KUKA KRL program: MyProgram_226().src

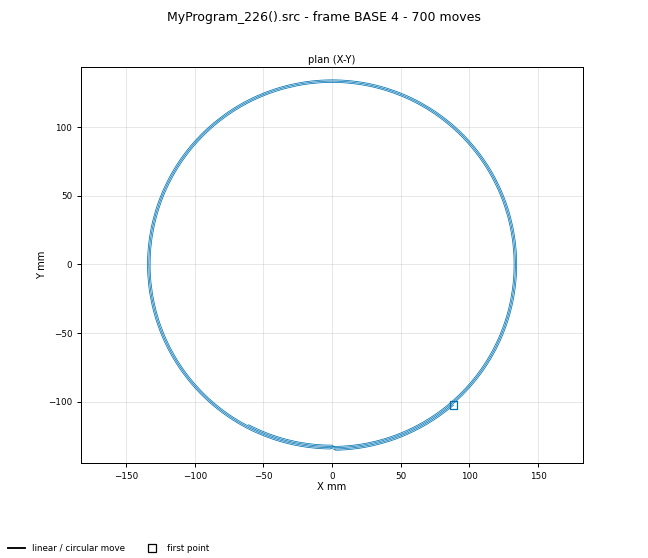
[picture p0: tool path of MyProgram_226().src in frame BASE 4, 700 of 700 moves have a stored position in this frame; points joined in program order, loops and branches not executed]
&ACCESS RVP
&REL 1
&PARAM TEMPLATE = C:\KRC\Roboter\Template\vorgabe
&PARAM EDITMASK = *
DEF MyProgram_226()
; ---- Setting reference (Base) ----
$BASE = BASE_DATA[4]

; --------------------------
; ---- Setting tool (TCP) ----
$TOOL = TOOL_DATA[3]
; --------------------------

$VEL.CP = VEL_APROX_PRINT
Startdeposition()
$VEL.CP = VEL_PRINT
LIN {X 88.4105,Y -102.4837,Z 156,A -52.8123,B 24.9683,C -1.3001,E1 25.1035,E2 499.4547} C_DIS
LIN {X 85.5901,Y -104.8506,Z 156,A -54.3172,B 24.9683,C -1.2995,E1 25.1003,E2 500.9552} C_DIS
LIN {X 81.9541,Y -107.7171,Z 156,A -56.2769,B 24.9686,C -1.2951,E1 25.096,E2 502.918} C_DIS
LIN {X 78.4285,Y -110.3106,Z 156,A -58.1174,B 24.9687,C -1.2919,E1 25.0918,E2 504.7597} C_DIS
LIN {X 75.1109,Y -112.5952,Z 156,A -59.7943,B 24.9688,C -1.2899,E1 25.0879,E2 506.4355} C_DIS
LIN {X 71.3717,Y -115.0019,Z 156,A -61.6528,B 24.969,C -1.2876,E1 25.0835,E2 508.2937} C_DIS
LIN {X 67.9053,Y -117.0821,Z 156,A -63.3421,B 24.969,C -1.2855,E1 25.0795,E2 509.9826} C_DIS
LIN {X 64.3345,Y -119.0819,Z 156,A -65.1517,B 24.9694,C -1.2782,E1 25.075,E2 511.8043} C_DIS
LIN {X 59.8875,Y -121.3766,Z 156,A -67.0719,B 24.9691,C -1.2855,E1 25.0703,E2 513.702} C_DIS
LIN {X 57.2409,Y -122.6479,Z 156,A -68.3239,B 24.9691,C -1.2829,E1 25.0671,E2 514.9567} C_DIS
LIN {X 53.5301,Y -124.3116,Z 156,A -70.0894,B 24.9694,C -1.2779,E1 25.0626,E2 516.7299} C_DIS
LIN {X 50.109,Y -125.7306,Z 156,A -71.756,B 24.9698,C -1.2701,E1 25.0582,E2 518.4109} C_DIS
LIN {X 45.2698,Y -127.5536,Z 156,A -73.8005,B 24.9696,C -1.275,E1 25.0529,E2 520.4396} C_DIS
LIN {X 42.4798,Y -128.5083,Z 156,A -75.0813,B 24.9697,C -1.2717,E1 25.0495,E2 521.7258} C_DIS
LIN {X 38.7522,Y -129.683,Z 156,A -76.6927,B 24.9697,C -1.272,E1 25.0452,E2 523.3335} C_DIS
LIN {X 33.3545,Y -131.173,Z 156,A -79.0675,B 24.9698,C -1.2692,E1 25.0388,E2 525.7112} C_DIS
LIN {X 30.1099,Y -131.9555,Z 156,A -80.5038,B 24.97,C -1.2665,E1 25.0349,E2 527.1518} C_DIS
LIN {X 26.6432,Y -132.6994,Z 156,A -82.044,B 24.9701,C -1.2631,E1 25.0307,E2 528.6983} C_DIS
LIN {X 22.4298,Y -133.4759,Z 156,A -83.877,B 24.9702,C -1.2605,E1 25.0256,E2 530.5353} C_DIS
LIN {X 18.3422,Y -134.1009,Z 156,A -85.6848,B 24.9704,C -1.2562,E1 25.0206,E2 532.3517} C_DIS
LIN {X 14.4718,Y -134.5715,Z 156,A -87.2354,B 24.9702,C -1.2606,E1 25.0163,E2 533.8908} C_DIS
LIN {X 10.295,Y -134.9561,Z 156,A -89.0367,B 24.9703,C -1.2583,E1 25.0113,E2 535.6965} C_DIS
LIN {X 6.6876,Y -135.1822,Z 156,A -90.5035,B 24.9703,C -1.261,E1 25.0072,E2 537.1563} C_DIS
LIN {X 2.7111,Y -135.3212,Z 156,A -92.2608,B 24.9704,C -1.2566,E1 25.0023,E2 538.9238} C_DIS
LIN {X 2.7111,Y -135.3212,Z 156,A -92.2608,B 24.9704,C -1.2566,E1 25.0023,E2 538.9238} C_DIS
Enddeposition()
LIN {X 0.9355,Y -134.409,Z 156,A -91.9033,B 23.562,C -1.0427,E1 23.5861,E2 538.9103} C_DIS
Startdeposition()
$VEL.CP = VEL_PRINT
LIN {X 4.9293,Y -134.3237,Z 156,A -90.1147,B 23.5618,C -1.0476,E1 23.5911,E2 537.11} C_DIS
LIN {X 8.6316,Y -134.1368,Z 156,A -88.4447,B 23.5616,C -1.0528,E1 23.5958,E2 535.4278} C_DIS
LIN {X 12.8622,Y -133.7968,Z 156,A -86.7417,B 23.5618,C -1.0483,E1 23.6005,E2 533.7369} C_DIS
LIN {X 17.0675,Y -133.3262,Z 156,A -84.913,B 23.5617,C -1.0507,E1 23.6056,E2 531.9039} C_DIS
LIN {X 20.2692,Y -132.8768,Z 156,A -83.6497,B 23.5619,C -1.0458,E1 23.609,E2 530.654} C_DIS
LIN {X 23.6425,Y -132.3179,Z 156,A -82.0981,B 23.5616,C -1.0517,E1 23.6133,E2 529.0893} C_DIS
LIN {X 27.7995,Y -131.5086,Z 156,A -80.2512,B 23.5615,C -1.0554,E1 23.6184,E2 527.2357} C_DIS
LIN {X 31.3885,Y -130.6971,Z 156,A -78.7676,B 23.5616,C -1.0525,E1 23.6224,E2 525.7614} C_DIS
LIN {X 37.2329,Y -129.1549,Z 156,A -76.2005,B 23.5616,C -1.0548,E1 23.6294,E2 523.193} C_DIS
LIN {X 41.5122,Y -127.844,Z 156,A -74.1617,B 23.5611,C -1.0638,E1 23.6348,E2 521.1358} C_DIS
LIN {X 45.1666,Y -126.5982,Z 156,A -72.4547,B 23.5609,C -1.0691,E1 23.6394,E2 519.4191} C_DIS
LIN {X 49.906,Y -124.8057,Z 156,A -70.4656,B 23.5612,C -1.0632,E1 23.6445,E2 517.4494} C_DIS
LIN {X 53.121,Y -123.4712,Z 156,A -69.0171,B 23.5612,C -1.0636,E1 23.6482,E2 516.0036} C_DIS
LIN {X 56.8828,Y -121.7847,Z 156,A -67.2053,B 23.5609,C -1.0692,E1 23.6528,E2 514.1828} C_DIS
LIN {X 60.3051,Y -120.1281,Z 156,A -65.5272,B 23.5607,C -1.0748,E1 23.657,E2 512.4955} C_DIS
LIN {X 63.8728,Y -118.27,Z 156,A -63.8371,B 23.5606,C -1.0765,E1 23.6612,E2 510.8063} C_DIS
LIN {X 67.8011,Y -116.0627,Z 156,A -61.9275,B 23.5605,C -1.0794,E1 23.6658,E2 508.8956} C_DIS
LIN {X 70.6321,Y -114.3619,Z 156,A -60.5125,B 23.5603,C -1.0824,E1 23.6692,E2 507.4778} C_DIS
LIN {X 74.425,Y -111.9304,Z 156,A -58.6117,B 23.5603,C -1.0852,E1 23.6737,E2 505.5767} C_DIS
LIN {X 78.0467,Y -109.4357,Z 156,A -56.7416,B 23.5601,C -1.0888,E1 23.6779,E2 503.7045} C_DIS
LIN {X 81.7345,Y -106.7094,Z 156,A -54.8243,B 23.56,C -1.091,E1 23.6822,E2 501.7892} C_DIS
LIN {X 85.2048,Y -103.9597,Z 156,A -53.1718,B 23.5603,C -1.0828,E1 23.6858,E2 500.1636} C_DIS
LIN {X 88.1779,Y -101.4502,Z 156,A -51.272,B 23.5596,C -1.0993,E1 23.6899,E2 498.2307} C_DIS
LIN {X 91.4896,Y -98.4739,Z 156,A -49.3955,B 23.5594,C -1.1027,E1 23.6937,E2 496.3539} C_DIS
LIN {X 94.6611,Y -95.4291,Z 156,A -47.7139,B 23.5597,C -1.0971,E1 23.697,E2 494.6937} C_DIS
LIN {X 97.4339,Y -92.597,Z 156,A -45.834,B 23.5591,C -1.1114,E1 23.7007,E2 492.7869} C_DIS
LIN {X 100.4874,Y -89.2739,Z 156,A -43.8982,B 23.5588,C -1.117,E1 23.7044,E2 490.8464} C_DIS
LIN {X 103.3752,Y -85.9131,Z 156,A -42.0362,B 23.5587,C -1.1205,E1 23.7077,E2 488.9846} C_DIS
LIN {X 105.5443,Y -83.234,Z 156,A -40.6446,B 23.5587,C -1.1203,E1 23.7101,E2 487.6004} C_DIS
LIN {X 108.2335,Y -79.7055,Z 156,A -38.3873,B 23.5575,C -1.1451,E1 23.714,E2 485.293} C_DIS
LIN {X 110.5538,Y -76.4555,Z 156,A -37.0233,B 23.5581,C -1.1318,E1 23.7161,E2 483.9693} C_DIS
LIN {X 112.6587,Y -73.3176,Z 156,A -35.4269,B 23.558,C -1.1356,E1 23.7185,E2 482.3719} C_DIS
LIN {X 115.0279,Y -69.5415,Z 156,A -33.5351,B 23.5577,C -1.1407,E1 23.7213,E2 480.4778} C_DIS
LIN {X 117.3269,Y -65.5891,Z 156,A -31.5842,B 23.5575,C -1.1465,E1 23.724,E2 478.5232} C_DIS
LIN {X 119.5762,Y -61.3894,Z 156,A -29.6624,B 23.5575,C -1.1468,E1 23.7265,E2 476.6115} C_DIS
LIN {X 121.1879,Y -58.1416,Z 156,A -28.1905,B 23.5575,C -1.1475,E1 23.7283,E2 475.1462} C_DIS
LIN {X 122.593,Y -55.1176,Z 156,A -26.9535,B 23.5577,C -1.142,E1 23.7297,E2 473.93} C_DIS
LIN {X 124.1713,Y -51.4639,Z 156,A -25.0102,B 23.5568,C -1.1604,E1 23.7319,E2 471.9523} C_DIS
LIN {X 125.5328,Y -48.0514,Z 156,A -23.4937,B 23.5568,C -1.1626,E1 23.7334,E2 470.4393} C_DIS
LIN {X 126.9947,Y -44.0372,Z 156,A -21.7357,B 23.5566,C -1.165,E1 23.7351,E2 468.6858} C_DIS
LIN {X 128.2984,Y -40.0882,Z 156,A -19.7977,B 23.5559,C -1.1795,E1 23.7367,E2 466.7237} C_DIS
LIN {X 129.3686,Y -36.4803,Z 156,A -18.3244,B 23.556,C -1.1776,E1 23.7379,E2 465.264} C_DIS
LIN {X 130.2418,Y -33.2273,Z 156,A -16.9031,B 23.5558,C -1.1815,E1 23.7389,E2 463.8419} C_DIS
LIN {X 131.0539,Y -29.8641,Z 156,A -15.439,B 23.5556,C -1.1856,E1 23.7398,E2 462.3765} C_DIS
LIN {X 131.8298,Y -26.2341,Z 156,A -13.7478,B 23.5551,C -1.1966,E1 23.7408,E2 460.6685} C_DIS
LIN {X 132.5689,Y -22.1919,Z 156,A -12.1079,B 23.5551,C -1.1963,E1 23.7416,E2 459.0396} C_DIS
LIN {X 133.1787,Y -18.1926,Z 156,A -10.3049,B 23.5547,C -1.2061,E1 23.7423,E2 457.2235} C_DIS
LIN {X 133.636,Y -14.4372,Z 156,A -8.8205,B 23.5547,C -1.2046,E1 23.7427,E2 455.7524} C_DIS
LIN {X 133.9718,Y -10.8981,Z 156,A -7.1925,B 23.5542,C -1.2155,E1 23.7431,E2 454.1074} C_DIS
LIN {X 134.2369,Y -6.8942,Z 156,A -5.5996,B 23.5542,C -1.2148,E1 23.7434,E2 452.5263} C_DIS
LIN {X 134.3785,Y -3.1364,Z 156,A -3.9402,B 23.5538,C -1.2231,E1 23.7435,E2 450.8569} C_DIS
LIN {X 134.4111,Y 0.902,Z 156,A -2.2554,B 23.5537,C -1.2268,E1 23.7435,E2 449.1737} C_DIS
LIN {X 134.3168,Y 5.1048,Z 156,A -0.5175,B 23.5535,C -1.2297,E1 23.7434,E2 447.4395} C_DIS
LIN {X 134.1212,Y 8.8838,Z 156,A 1.1946,B 23.553,C -1.2402,E1 23.7431,E2 445.7121} C_DIS
LIN {X 133.7965,Y 12.8654,Z 156,A 2.7809,B 23.553,C -1.2395,E1 23.7427,E2 444.1376} C_DIS
LIN {X 133.3513,Y 16.8762,Z 156,A 4.5475,B 23.5526,C -1.2475,E1 23.7421,E2 442.3623} C_DIS
LIN {X 132.8369,Y 20.5268,Z 156,A 6.0461,B 23.5526,C -1.2487,E1 23.7415,E2 440.8702} C_DIS
LIN {X 132.2011,Y 24.2952,Z 156,A 7.7773,B 23.552,C -1.2593,E1 23.7407,E2 439.1234} C_DIS
LIN {X 131.4551,Y 28.0471,Z 156,A 9.2523,B 23.5522,C -1.2562,E1 23.7398,E2 437.6653} C_DIS
LIN {X 130.6957,Y 31.3946,Z 156,A 10.6789,B 23.5521,C -1.2588,E1 23.7389,E2 436.241} C_DIS
LIN {X 129.9072,Y 34.5123,Z 156,A 12.0302,B 23.5519,C -1.2621,E1 23.738,E2 434.89} C_DIS
LIN {X 129.2093,Y 37.047,Z 156,A 13.706,B 23.5502,C -1.2951,E1 23.7367,E2 433.1422} C_DIS
LIN {X 127.9487,Y 41.1844,Z 156,A 14.7255,B 23.5522,C -1.2569,E1 23.7359,E2 432.224} C_DIS
LIN {X 126.7506,Y 44.7415,Z 156,A 16.7516,B 23.5508,C -1.2842,E1 23.734,E2 430.1421} C_DIS
LIN {X 125.3854,Y 48.4304,Z 156,A 18.2968,B 23.5508,C -1.2823,E1 23.7325,E2 428.6109} C_DIS
LIN {X 124.1199,Y 51.5871,Z 156,A 19.712,B 23.5508,C -1.2847,E1 23.731,E2 427.1979} C_DIS
LIN {X 122.823,Y 54.6032,Z 156,A 21.1009,B 23.5506,C -1.2883,E1 23.7294,E2 425.8083} C_DIS
LIN {X 121.7454,Y 56.9678,Z 156,A 23.4055,B 23.547,C -1.3553,E1 23.7265,E2 423.35} C_DIS
LIN {X 118.1,Y 64.1862,Z 156,A 25.5319,B 23.5502,C -1.2944,E1 23.7239,E2 421.3872} C_DIS
LIN {X 116.0778,Y 67.7754,Z 156,A 27.5088,B 23.5494,C -1.3109,E1 23.7211,E2 419.3803} C_DIS
LIN {X 113.7505,Y 71.6121,Z 156,A 29.3824,B 23.5492,C -1.3139,E1 23.7184,E2 417.5092} C_DIS
LIN {X 110.4427,Y 76.6151,Z 156,A 31.878,B 23.549,C -1.3174,E1 23.7145,E2 415.0183} C_DIS
LIN {X 108.0404,Y 79.9678,Z 156,A 33.7103,B 23.5486,C -1.3257,E1 23.7114,E2 413.1747} C_DIS
LIN {X 105.3495,Y 83.4805,Z 156,A 35.5509,B 23.5485,C -1.3279,E1 23.7083,E2 411.3378} C_DIS
LIN {X 102.5498,Y 86.8966,Z 156,A 37.4338,B 23.5482,C -1.3324,E1 23.7049,E2 409.453} C_DIS
LIN {X 99.5207,Y 90.3496,Z 156,A 39.3668,B 23.5481,C -1.3357,E1 23.7013,E2 407.5211} C_DIS
LIN {X 96.3825,Y 93.6905,Z 156,A 41.326,B 23.5478,C -1.3403,E1 23.6975,E2 405.5594} C_DIS
LIN {X 93.1606,Y 96.8953,Z 156,A 43.2788,B 23.5476,C -1.3452,E1 23.6936,E2 403.603} C_DIS
LIN {X 89.8181,Y 100.0009,Z 156,A 45.1818,B 23.5475,C -1.3471,E1 23.6897,E2 401.7036} C_DIS
LIN {X 86.5112,Y 102.875,Z 156,A 47.1668,B 23.5469,C -1.3569,E1 23.6855,E2 399.7025} C_DIS
LIN {X 82.6643,Y 105.9916,Z 156,A 49.1771,B 23.5469,C -1.3556,E1 23.6811,E2 397.7033} C_DIS
LIN {X 79.0174,Y 108.7368,Z 156,A 51.0711,B 23.5469,C -1.3564,E1 23.6768,E2 395.8145} C_DIS
LIN {X 75.3974,Y 111.2774,Z 156,A 52.9361,B 23.5469,C -1.3586,E1 23.6726,E2 393.9509} C_DIS
LIN {X 71.6195,Y 113.7458,Z 156,A 54.8649,B 23.5467,C -1.362,E1 23.668,E2 392.0204} C_DIS
LIN {X 64.5776,Y 117.8865,Z 156,A 58.129,B 23.547,C -1.3559,E1 23.6602,E2 388.7821} C_DIS
LIN {X 61.6399,Y 119.4486,Z 156,A 59.7847,B 23.5462,C -1.3699,E1 23.656,E2 387.0963} C_DIS
LIN {X 58.2078,Y 121.1563,Z 156,A 61.3017,B 23.5464,C -1.366,E1 23.6523,E2 385.5933} C_DIS
LIN {X 55.0775,Y 122.6109,Z 156,A 62.715,B 23.5464,C -1.3648,E1 23.6487,E2 384.1868} C_DIS
LIN {X 52.0438,Y 123.9292,Z 156,A 64.1422,B 23.5464,C -1.3673,E1 23.645,E2 382.7571} C_DIS
LIN {X 48.927,Y 125.1924,Z 156,A 65.5554,B 23.5464,C -1.3677,E1 23.6414,E2 381.3461} C_DIS
LIN {X 45.7794,Y 126.3773,Z 156,A 67.0293,B 23.5462,C -1.3711,E1 23.6375,E2 379.8671} C_DIS
LIN {X 40.214,Y 128.2587,Z 156,A 69.7843,B 23.5453,C -1.3859,E1 23.6301,E2 377.0809} C_DIS
LIN {X 35.0331,Y 129.7683,Z 156,A 71.8583,B 23.5459,C -1.3761,E1 23.6246,E2 375.0349} C_DIS
LIN {X 31.8551,Y 130.5847,Z 156,A 73.1872,B 23.546,C -1.3734,E1 23.621,E2 373.7147} C_DIS
LIN {X 28.4733,Y 131.3631,Z 156,A 74.6442,B 23.546,C -1.3731,E1 23.617,E2 372.2606} C_DIS
LIN {X 25.2847,Y 132.0139,Z 156,A 76.1047,B 23.5458,C -1.3774,E1 23.613,E2 370.7913} C_DIS
LIN {X 21.4016,Y 132.7008,Z 156,A 77.8884,B 23.5455,C -1.3831,E1 23.6081,E2 368.9953} C_DIS
LIN {X 17.7692,Y 133.2342,Z 156,A 79.3076,B 23.5459,C -1.3763,E1 23.6042,E2 367.5944} C_DIS
LIN {X 14.414,Y 133.6385,Z 156,A 80.769,B 23.5458,C -1.3776,E1 23.6001,E2 366.1308} C_DIS
LIN {X 10.5207,Y 134.0033,Z 156,A 82.5503,B 23.5455,C -1.3834,E1 23.5951,E2 364.3361} C_DIS
LIN {X 6.6231,Y 134.2505,Z 156,A 84.1088,B 23.5458,C -1.3782,E1 23.5908,E2 362.7913} C_DIS
LIN {X 2.6276,Y 134.3887,Z 156,A 85.8422,B 23.5457,C -1.3795,E1 23.586,E2 361.0551} C_DIS
LIN {X -1.2006,Y 134.4092,Z 156,A 87.5342,B 23.5455,C -1.3821,E1 23.5812,E2 359.3564} C_DIS
LIN {X -5.1809,Y 134.3139,Z 156,A 89.1183,B 23.5459,C -1.3761,E1 23.5769,E2 357.7872} C_DIS
LIN {X -8.9337,Y 134.1182,Z 156,A 90.842,B 23.5456,C -1.3814,E1 23.572,E2 356.0495} C_DIS
LIN {X -12.5875,Y 133.8232,Z 156,A 92.3234,B 23.5458,C -1.3768,E1 23.5679,E2 354.5791} C_DIS
LIN {X -16.2078,Y 133.4332,Z 156,A 93.9451,B 23.5458,C -1.3793,E1 23.5634,E2 352.95} C_DIS
LIN {X -20.4166,Y 132.854,Z 156,A 95.6742,B 23.546,C -1.3741,E1 23.5587,E2 351.2322} C_DIS
LIN {X -23.4422,Y 132.3537,Z 156,A 97.0071,B 23.546,C -1.3744,E1 23.555,E2 349.8972} C_DIS
LIN {X -26.9161,Y 131.691,Z 156,A 98.5253,B 23.546,C -1.3737,E1 23.5508,E2 348.3789} C_DIS
LIN {X -31.1661,Y 130.7508,Z 156,A 100.375,B 23.5461,C -1.3718,E1 23.5458,E2 346.5317} C_DIS
LIN {X -34.6648,Y 129.8665,Z 156,A 101.8848,B 23.5463,C -1.3689,E1 23.5417,E2 345.0267} C_DIS
LIN {X -37.9523,Y 128.9442,Z 156,A 103.3552,B 23.5463,C -1.368,E1 23.5378,E2 343.5559} C_DIS
LIN {X -41.897,Y 127.7182,Z 156,A 105.2086,B 23.5462,C -1.3704,E1 23.5328,E2 341.693} C_DIS
LIN {X -45.4507,Y 126.4958,Z 156,A 106.7099,B 23.5466,C -1.3636,E1 23.5289,E2 340.2057} C_DIS
LIN {X -48.5064,Y 125.3559,Z 156,A 108.1017,B 23.5466,C -1.3618,E1 23.5253,E2 338.8152} C_DIS
LIN {X -51.7489,Y 124.0523,Z 156,A 109.5956,B 23.5468,C -1.3599,E1 23.5214,E2 337.3225} C_DIS
LIN {X -54.6578,Y 122.7986,Z 156,A 110.9774,B 23.5468,C -1.3594,E1 23.5179,E2 335.9384} C_DIS
LIN {X -57.7764,Y 121.3624,Z 156,A 112.4472,B 23.5468,C -1.3575,E1 23.5142,E2 334.4695} C_DIS
LIN {X -60.8761,Y 119.8374,Z 156,A 113.9277,B 23.547,C -1.3554,E1 23.5105,E2 332.9899} C_DIS
LIN {X -64.2136,Y 118.085,Z 156,A 115.6185,B 23.547,C -1.3567,E1 23.5063,E2 331.2909} C_DIS
LIN {X -68.1273,Y 115.8711,Z 156,A 117.6526,B 23.5468,C -1.3588,E1 23.5014,E2 329.2449} C_DIS
LIN {X -72.3832,Y 113.2613,Z 156,A 119.6227,B 23.5474,C -1.3473,E1 23.4967,E2 327.2971} C_DIS
LIN {X -75.7909,Y 111.0103,Z 156,A 121.4528,B 23.5474,C -1.3481,E1 23.4925,E2 325.4586} C_DIS
LIN {X -78.3964,Y 109.1856,Z 156,A 122.943,B 23.5472,C -1.3517,E1 23.4891,E2 323.9538} C_DIS
LIN {X -86.439,Y 102.9355,Z 156,A 127.1437,B 23.5481,C -1.3355,E1 23.48,E2 319.7771} C_DIS
LIN {X -91.3964,Y 98.5606,Z 156,A 130.6218,B 23.5467,C -1.3602,E1 23.4726,E2 316.2221} C_DIS
LIN {X -95.3774,Y 94.7131,Z 156,A 132.2227,B 23.549,C -1.3186,E1 23.4696,E2 314.7185} C_DIS
LIN {X -100.4324,Y 89.3361,Z 156,A 135.7402,B 23.5485,C -1.328,E1 23.4629,E2 311.1607} C_DIS
LIN {X -102.6159,Y 86.8188,Z 156,A 136.9028,B 23.5493,C -1.3123,E1 23.4608,E2 310.0322} C_DIS
LIN {X -105.0907,Y 83.8056,Z 156,A 138.9915,B 23.5485,C -1.3278,E1 23.4571,E2 307.8938} C_DIS
LIN {X -107.634,Y 80.5136,Z 156,A 140.4229,B 23.5496,C -1.307,E1 23.4548,E2 306.5075} C_DIS
LIN {X -110.2504,Y 76.8916,Z 156,A 142.3253,B 23.5499,C -1.3016,E1 23.4517,E2 304.6087} C_DIS
LIN {X -112.7764,Y 73.1363,Z 156,A 144.2417,B 23.5502,C -1.2956,E1 23.4488,E2 302.6972} C_DIS
LIN {X -115.1894,Y 69.2744,Z 156,A 146.238,B 23.5503,C -1.2926,E1 23.4458,E2 300.6976} C_DIS
LIN {X -117.4617,Y 65.3472,Z 156,A 148.1357,B 23.5507,C -1.2852,E1 23.4432,E2 298.8077} C_DIS
LIN {X -118.9141,Y 62.6609,Z 156,A 149.5103,B 23.5507,C -1.2848,E1 23.4414,E2 297.4264} C_DIS
LIN {X -121.4329,Y 57.6288,Z 156,A 151.8272,B 23.5513,C -1.2737,E1 23.4386,E2 295.124} C_DIS
LIN {X -123.2208,Y 53.7001,Z 156,A 153.7306,B 23.5514,C -1.2711,E1 23.4364,E2 293.2162} C_DIS
LIN {X -124.6769,Y 50.2253,Z 156,A 155.2304,B 23.5519,C -1.2612,E1 23.4349,E2 291.7323} C_DIS
LIN {X -125.8009,Y 47.3402,Z 156,A 156.5728,B 23.5521,C -1.2581,E1 23.4335,E2 290.3895} C_DIS
LIN {X -127.1714,Y 43.5276,Z 156,A 158.8466,B 23.5511,C -1.2781,E1 23.4314,E2 288.0517} C_DIS
LIN {X -128.5083,Y 39.4029,Z 156,A 160.097,B 23.5528,C -1.2445,E1 23.4304,E2 286.8781} C_DIS
LIN {X -129.8132,Y 34.8649,Z 156,A 162.2281,B 23.5528,C -1.2435,E1 23.4288,E2 284.7363} C_DIS
LIN {X -130.5027,Y 32.1952,Z 156,A 163.3542,B 23.5531,C -1.2374,E1 23.428,E2 283.6185} C_DIS
LIN {X -131.6858,Y 26.9419,Z 156,A 165.6899,B 23.5534,C -1.2319,E1 23.4266,E2 281.2821} C_DIS
LIN {X -132.2816,Y 23.8455,Z 156,A 167.0534,B 23.5536,C -1.2284,E1 23.4259,E2 279.9187} C_DIS
LIN {X -132.829,Y 20.5784,Z 156,A 168.4865,B 23.5538,C -1.2248,E1 23.4253,E2 278.4855} C_DIS
LIN {X -133.3013,Y 17.2573,Z 156,A 169.9458,B 23.5539,C -1.2215,E1 23.4248,E2 277.0253} C_DIS
LIN {X -133.7537,Y 13.311,Z 156,A 171.736,B 23.5539,C -1.2205,E1 23.4242,E2 275.2262} C_DIS
LIN {X -134.0853,Y 9.3983,Z 156,A 173.4348,B 23.5542,C -1.2162,E1 23.4239,E2 273.5274} C_DIS
LIN {X -134.3113,Y 5.247,Z 156,A 175.1399,B 23.5546,C -1.2073,E1 23.4236,E2 271.8337} C_DIS
LIN {X -134.4101,Y 1.1043,Z 156,A 176.9758,B 23.5547,C -1.2047,E1 23.4236,E2 269.9924} C_DIS
LIN {X -134.3738,Y -3.3067,Z 156,A 178.8659,B 23.555,C -1.1991,E1 23.4236,E2 268.1044} C_DIS
LIN {X -134.21,Y -7.4289,Z 156,A -179.336,B 23.5552,C -1.1952,E1 23.4239,E2 266.3045} C_DIS
LIN {X -133.9579,Y -11.0623,Z 156,A -177.9212,B 23.5557,C -1.1838,E1 23.4242,E2 264.9093} C_DIS
LIN {X -133.67,Y -14.1212,Z 156,A -176.5911,B 23.5559,C -1.1805,E1 23.4246,E2 263.5789} C_DIS
LIN {X -133.2726,Y -17.4761,Z 156,A -175.1064,B 23.556,C -1.178,E1 23.4251,E2 262.091} C_DIS
LIN {X -132.7171,Y -21.3009,Z 156,A -173.3744,B 23.556,C -1.1766,E1 23.4258,E2 260.3515} C_DIS
LIN {X -130.971,Y -30.2267,Z 156,A -169.4419,B 23.5565,C -1.1669,E1 23.428,E2 256.4187} C_DIS
LIN {X -129.9653,Y -34.2942,Z 156,A -167.5966,B 23.5567,C -1.1641,E1 23.4293,E2 254.5689} C_DIS
LIN {X -128.6367,Y -38.9832,Z 156,A -165.6294,B 23.5572,C -1.1526,E1 23.4308,E2 252.6185} C_DIS
LIN {X -127.5991,Y -42.2547,Z 156,A -164.1865,B 23.5574,C -1.1472,E1 23.4321,E2 251.1803} C_DIS
LIN {X -126.5615,Y -45.2685,Z 156,A -162.7938,B 23.5576,C -1.1447,E1 23.4334,E2 249.7855} C_DIS
LIN {X -125.3591,Y -48.4981,Z 156,A -161.3418,B 23.5578,C -1.1395,E1 23.4348,E2 248.3377} C_DIS
LIN {X -124.1029,Y -51.6277,Z 156,A -159.8952,B 23.558,C -1.1357,E1 23.4363,E2 246.8921} C_DIS
LIN {X -122.7509,Y -54.7644,Z 156,A -158.427,B 23.5581,C -1.1321,E1 23.438,E2 245.4245} C_DIS
LIN {X -121.3559,Y -57.7899,Z 156,A -157.1312,B 23.5586,C -1.1222,E1 23.4395,E2 244.146} C_DIS
LIN {X -119.8283,Y -60.894,Z 156,A -155.5341,B 23.5586,C -1.1238,E1 23.4415,E2 242.5358} C_DIS
LIN {X -118.182,Y -64.0359,Z 156,A -153.8691,B 23.5584,C -1.1267,E1 23.4437,E2 240.8538} C_DIS
LIN {X -115.9859,Y -67.9318,Z 156,A -151.9715,B 23.5586,C -1.1211,E1 23.4463,E2 238.9598} C_DIS
LIN {X -113.6905,Y -71.7071,Z 156,A -150.0893,B 23.5589,C -1.1161,E1 23.4491,E2 237.0801} C_DIS
LIN {X -111.2697,Y -75.4088,Z 156,A -148.1853,B 23.559,C -1.112,E1 23.452,E2 235.176} C_DIS
LIN {X -108.6438,Y -79.1458,Z 156,A -146.2276,B 23.5592,C -1.1076,E1 23.4552,E2 233.2192} C_DIS
LIN {X -105.3039,Y -83.5378,Z 156,A -143.7669,B 23.5592,C -1.107,E1 23.4595,E2 230.7475} C_DIS
LIN {X -102.7175,Y -86.6989,Z 156,A -142.0676,B 23.5595,C -1.1009,E1 23.4625,E2 229.0553} C_DIS
LIN {X -99.7538,Y -90.0928,Z 156,A -140.1461,B 23.5597,C -1.0965,E1 23.466,E2 227.1356} C_DIS
LIN {X -96.6276,Y -93.4373,Z 156,A -138.25,B 23.56,C -1.0896,E1 23.4697,E2 225.2482} C_DIS
LIN {X -93.5068,Y -96.5605,Z 156,A -136.2778,B 23.56,C -1.0899,E1 23.4736,E2 223.2664} C_DIS
LIN {X -90.0096,Y -99.8292,Z 156,A -134.2737,B 23.5603,C -1.0839,E1 23.4777,E2 221.2685} C_DIS
LIN {X -86.6767,Y -102.7361,Z 156,A -132.3628,B 23.5603,C -1.0815,E1 23.4818,E2 219.3558} C_DIS
LIN {X -83.2189,Y -105.5561,Z 156,A -130.4522,B 23.5605,C -1.0783,E1 23.486,E2 217.4455} C_DIS
LIN {X -79.6785,Y -108.2533,Z 156,A -128.5631,B 23.5607,C -1.0746,E1 23.4902,E2 215.5587} C_DIS
LIN {X -75.9497,Y -110.9013,Z 156,A -126.6265,B 23.5608,C -1.0707,E1 23.4946,E2 213.6248} C_DIS
LIN {X -72.6562,Y -113.0865,Z 156,A -124.4093,B 23.5598,C -1.0939,E1 23.5,E2 211.3416} C_DIS
LIN {X -68.4589,Y -115.6762,Z 156,A -122.7757,B 23.561,C -1.0679,E1 23.5037,E2 209.7681} C_DIS
LIN {X -65.6597,Y -117.2872,Z 156,A -121.417,B 23.561,C -1.065,E1 23.507,E2 208.4122} C_DIS
LIN {X -61.4474,Y -119.5466,Z 156,A -119.4249,B 23.5613,C -1.0601,E1 23.5119,E2 206.4266} C_DIS
LIN {X -58.3216,Y -121.1019,Z 156,A -117.9448,B 23.5613,C -1.0579,E1 23.5157,E2 204.9479} C_DIS
LIN {X -55.0775,Y -122.6109,Z 156,A -116.4593,B 23.5615,C -1.0542,E1 23.5194,E2 203.4678} C_DIS
LIN {X -51.9501,Y -123.9683,Z 156,A -114.995,B 23.5615,C -1.0532,E1 23.5232,E2 202.0024} C_DIS
LIN {X -48.948,Y -125.1842,Z 156,A -113.6127,B 23.5616,C -1.0519,E1 23.5268,E2 200.6202} C_DIS
LIN {X -43.3287,Y -127.2404,Z 156,A -110.8203,B 23.5612,C -1.0615,E1 23.5342,E2 197.7978} C_DIS
LIN {X -38.4626,Y -128.7948,Z 156,A -108.7784,B 23.5616,C -1.0531,E1 23.5396,E2 195.7731} C_DIS
LIN {X -34.8536,Y -129.8162,Z 156,A -107.287,B 23.5619,C -1.0468,E1 23.5436,E2 194.2951} C_DIS
LIN {X -31.7292,Y -130.615,Z 156,A -105.9045,B 23.5619,C -1.0464,E1 23.5473,E2 192.9115} C_DIS
LIN {X -28.4249,Y -131.3736,Z 156,A -104.4485,B 23.5619,C -1.0462,E1 23.5513,E2 191.454} C_DIS
LIN {X -24.7544,Y -132.1153,Z 156,A -102.7313,B 23.5616,C -1.0516,E1 23.556,E2 189.7214} C_DIS
LIN {X -20.6359,Y -132.8201,Z 156,A -101.1051,B 23.562,C -1.0433,E1 23.5605,E2 188.1142} C_DIS
LIN {X -17.2421,Y -133.3033,Z 156,A -99.5981,B 23.562,C -1.0453,E1 23.5647,E2 186.6011} C_DIS
LIN {X -13.2467,Y -133.7599,Z 156,A -97.8558,B 23.5619,C -1.0465,E1 23.5695,E2 184.8547} C_DIS
LIN {X -9.6363,Y -134.0679,Z 156,A -96.3224,B 23.5619,C -1.0459,E1 23.5738,E2 183.3221} C_DIS
LIN {X -5.3887,Y -134.3058,Z 156,A -94.5268,B 23.5619,C -1.0451,E1 23.5788,E2 181.5281} C_DIS
LIN {X -1.4644,Y -134.4077,Z 156,A -92.7415,B 23.5617,C -1.051,E1 23.5838,E2 179.7279} C_DIS
LIN {X -1.4644,Y -134.4077,Z 156,A -92.7415,B 23.5617,C -1.051,E1 23.5838,E2 179.7279} C_DIS
Enddeposition()
LIN {X 0.9262,Y -133.4745,Z 156,A -91.6381,B 22.3243,C -0.839,E1 22.3412,E2 179.0215} C_DIS
Startdeposition()
$VEL.CP = VEL_PRINT
LIN {X -1.4317,Y -133.4741,Z 156,A -93.2247,B 22.3252,C -0.8117,E1 22.3366,E2 180.6798} C_DIS
LIN {X -5.2344,Y -133.3773,Z 156,A -94.7418,B 22.325,C -0.817,E1 22.3324,E2 182.1833} C_DIS
LIN {X -8.9431,Y -133.182,Z 156,A -96.4837,B 22.3253,C -0.8101,E1 22.3275,E2 183.9442} C_DIS
LIN {X -12.7579,Y -132.8688,Z 156,A -97.9962,B 22.3251,C -0.8163,E1 22.3233,E2 185.4411} C_DIS
LIN {X -16.1783,Y -132.4963,Z 156,A -99.4775,B 22.3251,C -0.8163,E1 22.3192,E2 186.9235} C_DIS
LIN {X -19.5244,Y -132.0457,Z 156,A -100.898,B 22.3251,C -0.818,E1 22.3153,E2 188.3409} C_DIS
LIN {X -22.424,Y -131.5835,Z 156,A -102.1695,B 22.3251,C -0.8179,E1 22.3118,E2 189.6139} C_DIS
LIN {X -25.5765,Y -131.0075,Z 156,A -103.5385,B 22.325,C -0.8187,E1 22.308,E2 190.9823} C_DIS
LIN {X -28.6252,Y -130.375,Z 156,A -104.903,B 22.325,C -0.818,E1 22.3043,E2 192.3505} C_DIS
LIN {X -32.0577,Y -129.5754,Z 156,A -106.3983,B 22.325,C -0.8196,E1 22.3002,E2 193.8438} C_DIS
LIN {X -35.1717,Y -128.765,Z 156,A -107.7834,B 22.325,C -0.8203,E1 22.2965,E2 195.2296} C_DIS
LIN {X -37.7619,Y -128.027,Z 156,A -108.9854,B 22.325,C -0.8191,E1 22.2932,E2 196.437} C_DIS
LIN {X -41.395,Y -126.9012,Z 156,A -110.5805,B 22.3249,C -0.822,E1 22.289,E2 198.0276} C_DIS
LIN {X -44.3694,Y -125.8913,Z 156,A -111.9335,B 22.3249,C -0.823,E1 22.2854,E2 199.381} C_DIS
LIN {X -47.3072,Y -124.8162,Z 156,A -113.2991,B 22.3249,C -0.8232,E1 22.2819,E2 200.7493} C_DIS
LIN {X -50.5447,Y -123.5414,Z 156,A -114.771,B 22.3247,C -0.8257,E1 22.2781,E2 202.2183} C_DIS
LIN {X -53.3009,Y -122.3761,Z 156,A -116.0706,B 22.3247,C -0.8264,E1 22.2747,E2 203.5194} C_DIS
LIN {X -56.603,Y -120.8854,Z 156,A -117.623,B 22.3247,C -0.8283,E1 22.2708,E2 205.0711} C_DIS
LIN {X -59.3938,Y -119.5378,Z 156,A -118.9724,B 22.3247,C -0.8291,E1 22.2674,E2 206.4225} C_DIS
LIN {X -62.6785,Y -117.8501,Z 156,A -120.5284,B 22.3245,C -0.8324,E1 22.2635,E2 207.9744} C_DIS
LIN {X -65.8321,Y -116.1187,Z 156,A -122.2431,B 22.3247,C -0.8269,E1 22.2593,E2 209.7094} C_DIS
LIN {X -69.4351,Y -114.001,Z 156,A -123.9086,B 22.3244,C -0.8353,E1 22.2554,E2 211.3585} C_DIS
LIN {X -72.7722,Y -111.8995,Z 156,A -125.6545,B 22.3244,C -0.8356,E1 22.2512,E2 213.1099} C_DIS
LIN {X -76.3801,Y -109.4687,Z 156,A -127.518,B 22.3243,C -0.8388,E1 22.2469,E2 214.972} C_DIS
LIN {X -79.6291,Y -107.1284,Z 156,A -129.3002,B 22.3243,C -0.839,E1 22.2429,E2 216.7609} C_DIS
LIN {X -82.9917,Y -104.5452,Z 156,A -131.1331,B 22.3242,C -0.8417,E1 22.2389,E2 218.5942} C_DIS
LIN {X -86.0704,Y -102.026,Z 156,A -132.7552,B 22.3239,C -0.8487,E1 22.2354,E2 220.2048} C_DIS
LIN {X -88.7329,Y -99.7193,Z 156,A -134.2747,B 22.3239,C -0.8514,E1 22.2322,E2 221.7241} C_DIS
LIN {X -91.5687,Y -97.1209,Z 156,A -135.999,B 22.3239,C -0.8515,E1 22.2287,E2 223.4559} C_DIS
LIN {X -94.3861,Y -94.3861,Z 156,A -137.6474,B 22.3236,C -0.8567,E1 22.2254,E2 225.0985} C_DIS
LIN {X -97.2347,Y -91.448,Z 156,A -139.4624,B 22.3236,C -0.858,E1 22.2219,E2 226.919} C_DIS
LIN {X -100.2435,Y -88.14,Z 156,A -141.3303,B 22.3233,C -0.8646,E1 22.2184,E2 228.7789} C_DIS
LIN {X -102.696,Y -85.2692,Z 156,A -143.0562,B 22.3233,C -0.8638,E1 22.2153,E2 230.5159} C_DIS
LIN {X -105.238,Y -82.1122,Z 156,A -144.6938,B 22.3231,C -0.8724,E1 22.2125,E2 232.1395} C_DIS
LIN {X -107.3188,Y -79.3734,Z 156,A -146.305,B 22.3231,C -0.8702,E1 22.2098,E2 233.7654} C_DIS
LIN {X -109.8141,Y -75.8837,Z 156,A -148.0299,B 22.3228,C -0.8799,E1 22.207,E2 235.4742} C_DIS
LIN {X -111.9668,Y -72.6686,Z 156,A -149.788,B 22.3228,C -0.8799,E1 22.2043,E2 237.2422} C_DIS
LIN {X -114.3949,Y -68.7837,Z 156,A -151.7485,B 22.3226,C -0.8854,E1 22.2014,E2 239.1996} C_DIS
LIN {X -116.569,Y -65.0317,Z 156,A -153.5563,B 22.3223,C -0.8927,E1 22.199,E2 240.9988} C_DIS
LIN {X -118.4036,Y -61.6245,Z 156,A -155.2508,B 22.3222,C -0.8958,E1 22.1967,E2 242.6951} C_DIS
LIN {X -120.0787,Y -58.2972,Z 156,A -156.8349,B 22.322,C -0.9009,E1 22.1948,E2 244.2755} C_DIS
LIN {X -121.294,Y -55.7193,Z 156,A -158.062,B 22.3219,C -0.9043,E1 22.1933,E2 245.5013} C_DIS
LIN {X -122.6189,Y -52.7395,Z 156,A -159.4865,B 22.3217,C -0.9072,E1 22.1917,E2 246.9269} C_DIS
LIN {X -123.9535,Y -49.5225,Z 156,A -160.9999,B 22.3217,C -0.9108,E1 22.1901,E2 248.4405} C_DIS
LIN {X -125.2403,Y -46.1749,Z 156,A -162.5291,B 22.3214,C -0.9157,E1 22.1886,E2 249.9663} C_DIS
LIN {X -126.6999,Y -41.9997,Z 156,A -164.4451,B 22.3212,C -0.9207,E1 22.1869,E2 251.8817} C_DIS
LIN {X -127.743,Y -38.7126,Z 156,A -165.951,B 22.3211,C -0.924,E1 22.1857,E2 253.3885} C_DIS
LIN {X -128.765,Y -35.1717,Z 156,A -167.515,B 22.3209,C -0.9296,E1 22.1845,E2 254.9481} C_DIS
LIN {X -129.4606,Y -32.5099,Z 156,A -168.7333,B 22.3208,C -0.9316,E1 22.1836,E2 256.169} C_DIS
LIN {X -130.2763,Y -29.0752,Z 156,A -170.2266,B 22.3206,C -0.9372,E1 22.1827,E2 257.6574} C_DIS
LIN {X -130.931,Y -25.9683,Z 156,A -171.597,B 22.3204,C -0.9411,E1 22.1819,E2 259.0267} C_DIS
LIN {X -131.5077,Y -22.8692,Z 156,A -172.9511,B 22.3202,C -0.9453,E1 22.1813,E2 260.3787} C_DIS
LIN {X -131.9584,Y -20.0984,Z 156,A -174.2088,B 22.3202,C -0.9469,E1 22.1807,E2 261.6408} C_DIS
LIN {X -132.432,Y -16.7047,Z 156,A -175.6532,B 22.3199,C -0.9527,E1 22.1802,E2 263.0797} C_DIS
LIN {X -132.7959,Y -13.5173,Z 156,A -177.0344,B 22.3198,C -0.9568,E1 22.1798,E2 264.4592} C_DIS
LIN {X -133.0704,Y -10.4753,Z 156,A -178.3531,B 22.3196,C -0.9607,E1 22.1795,E2 265.7767} C_DIS
LIN {X -133.3209,Y -6.5161,Z 156,A 179.8854,B 22.3195,C -0.9637,E1 22.1792,E2 267.5423} C_DIS
LIN {X -133.4492,Y -2.9628,Z 156,A 178.3996,B 22.3192,C -0.9703,E1 22.179,E2 269.0208} C_DIS
LIN {X -133.4816,Y 0,Z 156,A 177.1596,B 22.319,C -0.9757,E1 22.179,E2 270.2548} C_DIS
LIN {X -133.436,Y 3.4364,Z 156,A 175.5723,B 22.319,C -0.9757,E1 22.1791,E2 271.853} C_DIS
LIN {X -133.3063,Y 6.8069,Z 156,A 174.1467,B 22.3188,C -0.9813,E1 22.1793,E2 273.2735} C_DIS
LIN {X -133.1028,Y 10.0322,Z 156,A 172.7374,B 22.3186,C -0.9849,E1 22.1796,E2 274.6831} C_DIS
LIN {X -132.808,Y 13.3907,Z 156,A 171.3064,B 22.3184,C -0.9902,E1 22.1799,E2 276.1097} C_DIS
LIN {X -132.4639,Y 16.4498,Z 156,A 169.9741,B 22.3182,C -0.994,E1 22.1804,E2 277.441} C_DIS
LIN {X -132.0995,Y 19.1479,Z 156,A 168.7442,B 22.3182,C -0.9951,E1 22.1808,E2 278.6761} C_DIS
LIN {X -131.5307,Y 22.7406,Z 156,A 167.2179,B 22.3179,C -1.0016,E1 22.1815,E2 280.1957} C_DIS
LIN {X -130.9696,Y 25.7745,Z 156,A 165.8798,B 22.3178,C -1.0052,E1 22.1822,E2 281.533} C_DIS
LIN {X -130.3058,Y 28.9459,Z 156,A 164.4762,B 22.3176,C -1.0091,E1 22.1831,E2 282.9358} C_DIS
LIN {X -129.6488,Y 31.7531,Z 156,A 163.2494,B 22.3174,C -1.0135,E1 22.1838,E2 284.1591} C_DIS
LIN {X -128.9113,Y 34.6228,Z 156,A 161.8983,B 22.3174,C -1.0142,E1 22.1848,E2 285.5174} C_DIS
LIN {X -127.8738,Y 38.2852,Z 156,A 160.2972,B 22.3171,C -1.0207,E1 22.1861,E2 287.1118} C_DIS
LIN {X -126.9012,Y 41.395,Z 156,A 158.8863,B 22.3169,C -1.0245,E1 22.1873,E2 288.5217} C_DIS
LIN {X -125.9184,Y 44.2911,Z 156,A 157.5602,B 22.3168,C -1.028,E1 22.1885,E2 289.8471} C_DIS
LIN {X -124.8369,Y 47.252,Z 156,A 156.172,B 22.3167,C -1.0307,E1 22.1898,E2 291.2371} C_DIS
LIN {X -123.5414,Y 50.5447,Z 156,A 154.6619,B 22.3164,C -1.0357,E1 22.1914,E2 292.7435} C_DIS
LIN {X -122.2424,Y 53.6101,Z 156,A 153.2251,B 22.3163,C -1.0397,E1 22.193,E2 294.1788} C_DIS
LIN {X -120.8607,Y 56.6564,Z 156,A 151.7775,B 22.3161,C -1.0435,E1 22.1947,E2 295.6253} C_DIS
LIN {X -119.3965,Y 59.6803,Z 156,A 150.3392,B 22.3159,C -1.0479,E1 22.1964,E2 297.0606} C_DIS
LIN {X -117.8501,Y 62.6785,Z 156,A 149.0434,B 22.3154,C -1.0587,E1 22.1981,E2 298.3358} C_DIS
LIN {X -116.569,Y 65.0317,Z 156,A 147.616,B 22.3158,C -1.0501,E1 22.2,E2 299.7943} C_DIS
LIN {X -114.4049,Y 68.7672,Z 156,A 145.7015,B 22.3157,C -1.0528,E1 22.2028,E2 301.713} C_DIS
LIN {X -111.9888,Y 72.6346,Z 156,A 143.7886,B 22.3153,C -1.0602,E1 22.2056,E2 303.6172} C_DIS
LIN {X -109.681,Y 76.075,Z 156,A 141.9674,B 22.3153,C -1.0633,E1 22.2085,E2 305.4406} C_DIS
LIN {X -107.3611,Y 79.3159,Z 156,A 140.3458,B 22.3148,C -1.0717,E1 22.2111,E2 307.0488} C_DIS
LIN {X -104.8544,Y 82.6007,Z 156,A 138.5025,B 22.3148,C -1.0734,E1 22.2143,E2 308.8974} C_DIS
LIN {X -102.026,Y 86.0704,Z 156,A 136.634,B 22.3144,C -1.0807,E1 22.2176,E2 310.7566} C_DIS
LIN {X -99.7193,Y 88.7329,Z 156,A 135.1125,B 22.3143,C -1.0841,E1 22.2204,E2 312.2768} C_DIS
LIN {X -97.3902,Y 91.2831,Z 156,A 133.5486,B 22.3143,C -1.0843,E1 22.2234,E2 313.8481} C_DIS
LIN {X -94.3861,Y 94.3861,Z 156,A 131.7639,B 22.3139,C -1.0917,E1 22.2268,E2 315.6216} C_DIS
LIN {X -91.9633,Y 96.7479,Z 156,A 130.2961,B 22.3138,C -1.0945,E1 22.2298,E2 317.089} C_DIS
LIN {X -89.4291,Y 99.0952,Z 156,A 128.8056,B 22.3136,C -1.0976,E1 22.2329,E2 318.5783} C_DIS
LIN {X -86.5865,Y 101.5878,Z 156,A 127.0708,B 22.3136,C -1.0963,E1 22.2365,E2 320.324} C_DIS
LIN {X -83.463,Y 104.17,Z 156,A 125.4266,B 22.3133,C -1.1042,E1 22.2401,E2 321.9544} C_DIS
LIN {X -80.8057,Y 106.2443,Z 156,A 123.9727,B 22.3132,C -1.107,E1 22.2433,E2 323.407} C_DIS
LIN {X -77.9976,Y 108.3228,Z 156,A 122.3533,B 22.3132,C -1.1048,E1 22.247,E2 325.0387} C_DIS
LIN {X -74.3639,Y 110.8484,Z 156,A 120.4356,B 22.3132,C -1.1077,E1 22.2514,E2 326.9559} C_DIS
LIN {X -70.9453,Y 113.0671,Z 156,A 118.7957,B 22.3128,C -1.1158,E1 22.2552,E2 328.5805} C_DIS
LIN {X -67.9759,Y 114.8771,Z 156,A 117.2466,B 22.3128,C -1.116,E1 22.2589,E2 330.1344} C_DIS
LIN {X -64.3522,Y 116.9453,Z 156,A 115.5083,B 22.3125,C -1.1214,E1 22.2631,E2 331.8641} C_DIS
LIN {X -61.3076,Y 118.57,Z 156,A 114.0224,B 22.3124,C -1.1237,E1 22.2668,E2 333.3488} C_DIS
LIN {X -58.7983,Y 119.8315,Z 156,A 112.8138,B 22.3124,C -1.1255,E1 22.2698,E2 334.5562} C_DIS
LIN {X -55.6968,Y 121.3044,Z 156,A 111.3405,B 22.3122,C -1.1277,E1 22.2736,E2 336.0277} C_DIS
LIN {X -52.2071,Y 122.849,Z 156,A 109.6937,B 22.3122,C -1.1297,E1 22.2778,E2 337.6738} C_DIS
LIN {X -49.134,Y 124.1101,Z 156,A 108.265,B 22.312,C -1.1315,E1 22.2815,E2 339.1014} C_DIS
LIN {X -46.348,Y 125.1755,Z 156,A 106.9845,B 22.312,C -1.1331,E1 22.2848,E2 340.3805} C_DIS
LIN {X -42.9477,Y 126.3842,Z 156,A 105.4307,B 22.3119,C -1.1348,E1 22.2889,E2 341.9333} C_DIS
LIN {X -39.9699,Y 127.3565,Z 156,A 104.0803,B 22.3119,C -1.1361,E1 22.2925,E2 343.2831} C_DIS
LIN {X -35.8223,Y 128.583,Z 156,A 102.2259,B 22.3117,C -1.1382,E1 22.2975,E2 345.1354} C_DIS
LIN {X -32.5861,Y 129.4412,Z 156,A 100.7447,B 22.3117,C -1.1376,E1 22.3015,E2 346.6206} C_DIS
LIN {X -29.0752,Y 130.2763,Z 156,A 99.2372,B 22.3116,C -1.1408,E1 22.3056,E2 348.1218} C_DIS
LIN {X -26.395,Y 130.8442,Z 156,A 98.0145,B 22.3116,C -1.1397,E1 22.3089,E2 349.3491} C_DIS
LIN {X -22.8692,Y 131.5077,Z 156,A 96.5374,B 22.3114,C -1.1436,E1 22.313,E2 350.8175} C_DIS
LIN {X -20.2036,Y 131.9421,Z 156,A 95.3371,B 22.3114,C -1.1426,E1 22.3163,E2 352.0218} C_DIS
LIN {X -17.0587,Y 132.3856,Z 156,A 94.0109,B 22.3114,C -1.1451,E1 22.3199,E2 353.3426} C_DIS
LIN {X -13.5173,Y 132.7959,Z 156,A 92.4692,B 22.3114,C -1.1453,E1 22.3242,E2 354.8846} C_DIS
LIN {X -10.4753,Y 133.0704,Z 156,A 91.159,B 22.3114,C -1.1459,E1 22.3279,E2 356.194} C_DIS
LIN {X -6.2558,Y 133.334,Z 156,A 89.334,B 22.3114,C -1.1461,E1 22.3329,E2 358.019} C_DIS
LIN {X -2.4933,Y 133.457,Z 156,A 87.6612,B 22.3114,C -1.144,E1 22.3376,E2 359.6978} C_DIS
LIN {X 1.0723,Y 133.4761,Z 156,A 86.1675,B 22.3114,C -1.1459,E1 22.3418,E2 361.1863} C_DIS
LIN {X 5.0963,Y 133.3827,Z 156,A 84.4494,B 22.3113,C -1.1465,E1 22.3466,E2 362.9025} C_DIS
LIN {X 8.1886,Y 133.2285,Z 156,A 83.1062,B 22.3113,C -1.1458,E1 22.3503,E2 364.2468} C_DIS
LIN {X 11.3089,Y 133,Z 156,A 81.7481,B 22.3113,C -1.145,E1 22.3541,E2 365.6063} C_DIS
LIN {X 14.9181,Y 132.6451,Z 156,A 80.2339,B 22.3113,C -1.1467,E1 22.3583,E2 367.1149} C_DIS
LIN {X 18.1129,Y 132.2475,Z 156,A 78.8504,B 22.3113,C -1.1463,E1 22.3621,E2 368.4983} C_DIS
LIN {X 20.7486,Y 131.8577,Z 156,A 77.7192,B 22.3113,C -1.1465,E1 22.3652,E2 369.6276} C_DIS
LIN {X 23.7584,Y 131.3486,Z 156,A 76.3585,B 22.3114,C -1.1437,E1 22.369,E2 370.994} C_DIS
LIN {X 27.3918,Y 130.6413,Z 156,A 74.8048,B 22.3114,C -1.1445,E1 22.3732,E2 372.5434} C_DIS
LIN {X 30.5013,Y 129.9505,Z 156,A 73.4374,B 22.3114,C -1.1438,E1 22.377,E2 373.9106} C_DIS
LIN {X 33.1605,Y 129.2955,Z 156,A 72.2522,B 22.3114,C -1.1426,E1 22.3802,E2 375.0968} C_DIS
LIN {X 36.5993,Y 128.3657,Z 156,A 70.7285,B 22.3115,C -1.1418,E1 22.3843,E2 376.6199} C_DIS
LIN {X 39.4498,Y 127.5174,Z 156,A 69.4248,B 22.3116,C -1.1395,E1 22.3878,E2 377.9269} C_DIS
LIN {X 42.8187,Y 126.4271,Z 156,A 67.9413,B 22.3116,C -1.1399,E1 22.3917,E2 379.4061} C_DIS
LIN {X 45.9178,Y 125.3348,Z 156,A 66.5242,B 22.3116,C -1.1383,E1 22.3954,E2 380.8241} C_DIS
LIN {X 48.6278,Y 124.3069,Z 156,A 65.2928,B 22.3117,C -1.1377,E1 22.3986,E2 382.0542} C_DIS
LIN {X 51.7174,Y 123.0536,Z 156,A 63.8228,B 22.3119,C -1.1343,E1 22.4024,E2 383.5291} C_DIS
LIN {X 54.9947,Y 121.625,Z 156,A 62.3293,B 22.3119,C -1.1345,E1 22.4062,E2 385.018} C_DIS
LIN {X 58.0714,Y 120.1866,Z 156,A 60.8633,B 22.3119,C -1.1323,E1 22.4099,E2 386.4854} C_DIS
LIN {X 61.1828,Y 118.6335,Z 156,A 59.4535,B 22.3119,C -1.1343,E1 22.4134,E2 387.8857} C_DIS
LIN {X 65.7094,Y 116.1881,Z 156,A 57.1691,B 22.3122,C -1.1276,E1 22.419,E2 390.18} C_DIS
LIN {X 68.7672,Y 114.4049,Z 156,A 55.5259,B 22.3126,C -1.1195,E1 22.423,E2 391.8389} C_DIS
LIN {X 72.5328,Y 112.055,Z 156,A 53.6582,B 22.3126,C -1.1183,E1 22.4274,E2 393.7029} C_DIS
LIN {X 76.1879,Y 109.6024,Z 156,A 51.8159,B 22.3126,C -1.1173,E1 22.4317,E2 395.5406} C_DIS
LIN {X 79.5689,Y 107.1732,Z 156,A 49.9931,B 22.3129,C -1.1125,E1 22.4358,E2 397.3687} C_DIS
LIN {X 82.7329,Y 104.7505,Z 156,A 48.3945,B 22.3129,C -1.1147,E1 22.4393,E2 398.9549} C_DIS
LIN {X 85.4095,Y 102.5798,Z 156,A 46.9214,B 22.3129,C -1.1122,E1 22.4425,E2 400.4282} C_DIS
LIN {X 88.4148,Y 100.0005,Z 156,A 45.1645,B 22.3132,C -1.1061,E1 22.4462,E2 402.1933} C_DIS
LIN {X 91.3353,Y 97.341,Z 156,A 43.4178,B 22.3135,C -1.1001,E1 22.4498,E2 403.9476} C_DIS
LIN {X 94.3861,Y 94.3861,Z 156,A 41.6501,B 22.3135,C -1.0989,E1 22.4533,E2 405.71} C_DIS
LIN {X 97.341,Y 91.3353,Z 156,A 39.9136,B 22.3135,C -1.0991,E1 22.4566,E2 407.4376} C_DIS
LIN {X 99.6264,Y 88.8366,Z 156,A 38.4516,B 22.3137,C -1.0953,E1 22.4594,E2 408.9019} C_DIS
LIN {X 102.2348,Y 85.8214,Z 156,A 36.6937,B 22.314,C -1.0891,E1 22.4626,E2 410.6671} C_DIS
LIN {X 104.7063,Y 82.7892,Z 156,A 35.0266,B 22.3142,C -1.0856,E1 22.4655,E2 412.3344} C_DIS
LIN {X 107.2762,Y 79.4307,Z 156,A 33.2853,B 22.3142,C -1.0848,E1 22.4684,E2 414.0687} C_DIS
LIN {X 109.3246,Y 76.5872,Z 156,A 31.8052,B 22.3143,C -1.0821,E1 22.4708,E2 415.5475} C_DIS
LIN {X 111.2143,Y 73.816,Z 156,A 30.3408,B 22.3146,C -1.0772,E1 22.4731,E2 417.0165} C_DIS
LIN {X 113.5036,Y 70.2447,Z 156,A 28.5289,B 22.3148,C -1.0729,E1 22.4758,E2 418.8293} C_DIS
LIN {X 115.6978,Y 66.569,Z 156,A 26.6991,B 22.315,C -1.0683,E1 22.4784,E2 420.6604} C_DIS
LIN {X 117.7516,Y 62.8646,Z 156,A 24.9219,B 22.3151,C -1.0654,E1 22.4807,E2 422.4348} C_DIS
LIN {X 119.3346,Y 59.8056,Z 156,A 23.4618,B 22.3153,C -1.0621,E1 22.4826,E2 423.8946} C_DIS
LIN {X 120.8023,Y 56.7827,Z 156,A 22.0303,B 22.3154,C -1.0586,E1 22.4843,E2 425.3267} C_DIS
LIN {X 122.0795,Y 53.9787,Z 156,A 20.7257,B 22.3155,C -1.0557,E1 22.4858,E2 426.6307} C_DIS
LIN {X 123.3626,Y 50.9774,Z 156,A 19.3184,B 22.3157,C -1.0513,E1 22.4873,E2 428.0407} C_DIS
LIN {X 124.5275,Y 48.0603,Z 156,A 17.9943,B 22.3159,C -1.0486,E1 22.4887,E2 429.3636} C_DIS
LIN {X 125.6709,Y 44.9856,Z 156,A 16.5466,B 22.3161,C -1.0425,E1 22.4901,E2 430.8182} C_DIS
LIN {X 126.867,Y 41.4979,Z 156,A 15.0245,B 22.3162,C -1.0407,E1 22.4914,E2 432.3352} C_DIS
LIN {X 127.8464,Y 38.3747,Z 156,A 13.6315,B 22.3164,C -1.037,E1 22.4926,E2 433.7288} C_DIS
LIN {X 128.6282,Y 35.6606,Z 156,A 12.4132,B 22.3166,C -1.0331,E1 22.4935,E2 434.9496} C_DIS
LIN {X 129.5754,Y 32.0577,Z 156,A 10.8427,B 22.3167,C -1.0295,E1 22.4946,E2 436.5191} C_DIS
LIN {X 130.2763,Y 29.0752,Z 156,A 9.5395,B 22.3169,C -1.026,E1 22.4954,E2 437.8228} C_DIS
LIN {X 130.931,Y 25.9683,Z 156,A 8.2065,B 22.3169,C -1.0233,E1 22.4961,E2 439.1542} C_DIS
LIN {X 131.4384,Y 23.2562,Z 156,A 7.0331,B 22.3171,C -1.0201,E1 22.4967,E2 440.328} C_DIS
LIN {X 131.932,Y 20.269,Z 156,A 5.6881,B 22.3174,C -1.0138,E1 22.4973,E2 441.6807} C_DIS
LIN {X 132.432,Y 16.7047,Z 156,A 4.1924,B 22.3174,C -1.0113,E1 22.4979,E2 443.1729} C_DIS
LIN {X 132.7959,Y 13.5173,Z 156,A 2.8317,B 22.3177,C -1.0077,E1 22.4983,E2 444.5339} C_DIS
LIN {X 133.1501,Y 9.3837,Z 156,A 1.0576,B 22.3179,C -1.0024,E1 22.4987,E2 446.3099} C_DIS
LIN {X 133.3494,Y 5.9507,Z 156,A -0.5616,B 22.3184,C -0.9905,E1 22.4989,E2 447.9493} C_DIS
LIN {X 133.4634,Y 2.1096,Z 156,A -2.0489,B 22.3183,C -0.9933,E1 22.499,E2 449.4193} C_DIS
LIN {X 133.4718,Y -1.6015,Z 156,A -3.702,B 22.3186,C -0.9851,E1 22.499,E2 451.0826} C_DIS
LIN {X 133.3828,Y -5.0928,Z 156,A -5.1422,B 22.3186,C -0.9833,E1 22.4989,E2 452.518} C_DIS
LIN {X 133.2087,Y -8.5101,Z 156,A -6.5931,B 22.3188,C -0.9794,E1 22.4986,E2 453.9692} C_DIS
LIN {X 132.9528,Y -11.8678,Z 156,A -7.9997,B 22.319,C -0.9766,E1 22.4983,E2 455.3736} C_DIS
LIN {X 132.6958,Y -14.4474,Z 156,A -9.1031,B 22.319,C -0.9735,E1 22.498,E2 456.4777} C_DIS
LIN {X 132.3168,Y -17.5839,Z 156,A -10.4907,B 22.3193,C -0.9676,E1 22.4975,E2 457.8715} C_DIS
LIN {X 131.7886,Y -21.195,Z 156,A -12.0119,B 22.3195,C -0.9648,E1 22.4969,E2 459.3899} C_DIS
LIN {X 131.313,Y -23.9574,Z 156,A -13.2309,B 22.3196,C -0.9602,E1 22.4963,E2 460.6129} C_DIS
LIN {X 130.6413,Y -27.3918,Z 156,A -14.7012,B 22.3198,C -0.9569,E1 22.4955,E2 462.0819} C_DIS
LIN {X 129.6975,Y -31.551,Z 156,A -16.5307,B 22.32,C -0.9512,E1 22.4943,E2 463.9144} C_DIS
LIN {X 128.9259,Y -34.5681,Z 156,A -17.8786,B 22.3202,C -0.9464,E1 22.4933,E2 465.2661} C_DIS
LIN {X 127.9952,Y -37.8707,Z 156,A -19.34,B 22.3204,C -0.9423,E1 22.4922,E2 466.7286} C_DIS
LIN {X 126.9012,Y -41.395,Z 156,A -20.8887,B 22.3204,C -0.9391,E1 22.4909,E2 468.2759} C_DIS
LIN {X 125.9565,Y -44.1812,Z 156,A -22.1581,B 22.3207,C -0.9348,E1 22.4897,E2 469.5483} C_DIS
LIN {X 124.7096,Y -47.5919,Z 156,A -23.6935,B 22.3208,C -0.9312,E1 22.4882,E2 471.0835} C_DIS
LIN {X 123.5414,Y -50.5447,Z 156,A -25.0525,B 22.321,C -0.9272,E1 22.4868,E2 472.4444} C_DIS
LIN {X 122.2424,Y -53.6101,Z 156,A -26.4506,B 22.321,C -0.9244,E1 22.4853,E2 473.8412} C_DIS
LIN {X 120.9922,Y -56.3719,Z 156,A -27.7776,B 22.3213,C -0.9192,E1 22.4837,E2 475.1736} C_DIS
LIN {X 119.5342,Y -59.401,Z 156,A -29.2238,B 22.3215,C -0.9147,E1 22.4819,E2 476.6227} C_DIS
LIN {X 117.7849,Y -62.8027,Z 156,A -30.928,B 22.3218,C -0.9068,E1 22.4797,E2 478.3375} C_DIS
LIN {X 115.6978,Y -66.569,Z 156,A -32.8008,B 22.322,C -0.9002,E1 22.4771,E2 480.2165} C_DIS
LIN {X 113.5925,Y -70.101,Z 156,A -34.428,B 22.322,C -0.902,E1 22.4748,E2 481.8297} C_DIS
LIN {X 111.7239,Y -73.0427,Z 156,A -36.0209,B 22.3223,C -0.8929,E1 22.4724,E2 483.4371} C_DIS
LIN {X 109.2426,Y -76.7034,Z 156,A -37.9135,B 22.3225,C -0.888,E1 22.4694,E2 485.3321} C_DIS
LIN {X 106.8056,Y -80.0627,Z 156,A -39.5656,B 22.3225,C -0.8895,E1 22.4667,E2 486.9713} C_DIS
LIN {X 104.7063,Y -82.7892,Z 156,A -41.1627,B 22.3228,C -0.8796,E1 22.4639,E2 488.5857} C_DIS
LIN {X 101.8978,Y -86.2218,Z 156,A -43.0501,B 22.3229,C -0.8755,E1 22.4605,E2 490.4741} C_DIS
LIN {X 99.1434,Y -89.3759,Z 156,A -44.7139,B 22.3229,C -0.8775,E1 22.4574,E2 492.1243} C_DIS
LIN {X 96.4875,Y -92.2358,Z 156,A -46.442,B 22.3231,C -0.8707,E1 22.4541,E2 493.8615} C_DIS
LIN {X 93.6518,Y -95.1141,Z 156,A -48.2175,B 22.3234,C -0.8645,E1 22.4506,E2 495.6448} C_DIS
LIN {X 90.7036,Y -97.9299,Z 156,A -49.8443,B 22.3233,C -0.8664,E1 22.4473,E2 497.2591} C_DIS
LIN {X 88.14,Y -100.2435,Z 156,A -51.3457,B 22.3234,C -0.862,E1 22.4442,E2 498.765} C_DIS
LIN {X 84.9436,Y -102.9656,Z 156,A -53.1679,B 22.3236,C -0.8571,E1 22.4403,E2 500.5923} C_DIS
LIN {X 81.4886,Y -105.7214,Z 156,A -55.0053,B 22.3236,C -0.8559,E1 22.4362,E2 502.4251} C_DIS
LIN {X 78.6812,Y -107.8274,Z 156,A -56.4893,B 22.3237,C -0.8538,E1 22.4329,E2 503.9085} C_DIS
LIN {X 75.8837,Y -109.8141,Z 156,A -57.9545,B 22.3238,C -0.8512,E1 22.4296,E2 505.3747} C_DIS
LIN {X 72.8703,Y -111.8358,Z 156,A -59.6144,B 22.3241,C -0.8432,E1 22.4257,E2 507.0494} C_DIS
LIN {X 69.4351,Y -114.001,Z 156,A -61.2454,B 22.3241,C -0.8454,E1 22.4218,E2 508.6689} C_DIS
LIN {X 66.4508,Y -115.7657,Z 156,A -62.8619,B 22.3244,C -0.8365,E1 22.4179,E2 510.3031} C_DIS
LIN {X 62.8646,Y -117.7516,Z 156,A -64.4848,B 22.3242,C -0.84,E1 22.4139,E2 511.9113} C_DIS
LIN {X 60.0125,Y -119.2293,Z 156,A -65.8602,B 22.3243,C -0.8379,E1 22.4105,E2 513.288} C_DIS
LIN {X 56.7827,Y -120.8023,Z 156,A -67.3845,B 22.3243,C -0.8363,E1 22.4067,E2 514.812} C_DIS
LIN {X 54.1829,Y -121.9881,Z 156,A -68.5977,B 22.3244,C -0.8352,E1 22.4036,E2 516.0248} C_DIS
LIN {X 50.9739,Y -123.364,Z 156,A -70.1178,B 22.3245,C -0.832,E1 22.3997,E2 517.5492} C_DIS
LIN {X 47.72,Y -124.6597,Z 156,A -71.5943,B 22.3245,C -0.8312,E1 22.3958,E2 519.0241} C_DIS
LIN {X 44.9691,Y -125.6769,Z 156,A -72.8923,B 22.3247,C -0.8277,E1 22.3924,E2 520.3282} C_DIS
LIN {X 41.395,Y -126.9012,Z 156,A -74.4631,B 22.3247,C -0.8281,E1 22.3883,E2 521.8944} C_DIS
LIN {X 38.2852,Y -127.8738,Z 156,A -75.8561,B 22.3247,C -0.8268,E1 22.3845,E2 523.2882} C_DIS
LIN {X 35.1717,Y -128.765,Z 156,A -77.2411,B 22.3247,C -0.8255,E1 22.3808,E2 524.6738} C_DIS
LIN {X 32.2634,Y -129.5231,Z 156,A -78.5048,B 22.3247,C -0.8255,E1 22.3774,E2 525.9354} C_DIS
LIN {X 29.3216,Y -130.22,Z 156,A -79.827,B 22.3248,C -0.8231,E1 22.3738,E2 527.2618} C_DIS
LIN {X 25.9683,Y -130.931,Z 156,A -81.2847,B 22.3248,C -0.8225,E1 22.3698,E2 528.719} C_DIS
LIN {X 23.033,Y -131.4784,Z 156,A -82.5728,B 22.3249,C -0.8212,E1 22.3663,E2 530.0088} C_DIS
LIN {X 19.7805,Y -132.0076,Z 156,A -84.1138,B 22.3251,C -0.8142,E1 22.362,E2 531.5666} C_DIS
LIN {X 15.8934,Y -132.5303,Z 156,A -85.6671,B 22.325,C -0.8194,E1 22.3577,E2 533.105} C_DIS
LIN {X 12.6347,Y -132.8806,Z 156,A -87.0536,B 22.325,C -0.8196,E1 22.3538,E2 534.4899} C_DIS
LIN {X 9.645,Y -133.131,Z 156,A -88.352,B 22.325,C -0.8185,E1 22.3502,E2 535.7905} C_DIS
LIN {X 5.9507,Y -133.3494,Z 156,A -90.0584,B 22.3252,C -0.8123,E1 22.3454,E2 537.5124} C_DIS
LIN {X 2.205,Y -133.4618,Z 156,A -91.5777,B 22.3251,C -0.8161,E1 22.3412,E2 539.0215} C_DIS
LIN {X 2.205,Y -133.4618,Z 156,A -91.5777,B 22.3251,C -0.8161,E1 22.3412,E2 539.0215} C_DIS
Enddeposition()
LIN {X 0.9151,Y -132.5419,Z 156,A -91.2226,B 21.2699,C -0.6915,E1 21.2829,E2 538.8869} C_DIS
Startdeposition()
$VEL.CP = VEL_PRINT
LIN {X 4.8247,Y -132.4588,Z 156,A -89.4243,B 21.2697,C -0.6968,E1 21.288,E2 537.0743} C_DIS
LIN {X 8.5775,Y -132.269,Z 156,A -87.7284,B 21.2696,C -0.7007,E1 21.2927,E2 535.3686} C_DIS
LIN {X 12.6502,Y -131.9411,Z 156,A -86.0571,B 21.2696,C -0.6972,E1 21.2973,E2 533.7079} C_DIS
LIN {X 16.7764,Y -131.4808,Z 156,A -84.219,B 21.2696,C -0.7002,E1 21.3024,E2 531.8632} C_DIS
LIN {X 20.8197,Y -130.9014,Z 156,A -82.5903,B 21.2697,C -0.6952,E1 21.3069,E2 530.2502} C_DIS
LIN {X 24.2612,Y -130.3083,Z 156,A -80.8547,B 21.2694,C -0.7066,E1 21.3117,E2 528.4855} C_DIS
LIN {X 28.2297,Y -129.5051,Z 156,A -79.3009,B 21.2696,C -0.6992,E1 21.3159,E2 526.9545} C_DIS
LIN {X 31.1189,Y -128.8411,Z 156,A -77.9971,B 21.2696,C -0.7014,E1 21.3195,E2 525.6468} C_DIS
LIN {X 34.8061,Y -127.8961,Z 156,A -76.2089,B 21.2693,C -0.7096,E1 21.3244,E2 523.8395} C_DIS
LIN {X 38.6077,Y -126.7986,Z 156,A -74.4743,B 21.2692,C -0.7126,E1 21.329,E2 522.1002} C_DIS
LIN {X 42.3517,Y -125.5985,Z 156,A -72.9607,B 21.2694,C -0.7061,E1 21.333,E2 520.6081} C_DIS
LIN {X 46.1072,Y -124.2686,Z 156,A -71.0805,B 21.2691,C -0.7155,E1 21.338,E2 518.7064} C_DIS
LIN {X 50.244,Y -122.6558,Z 156,A -69.3468,B 21.2693,C -0.7096,E1 21.3424,E2 516.9939} C_DIS
LIN {X 52.9273,Y -121.5204,Z 156,A -68.0912,B 21.2693,C -0.7113,E1 21.3456,E2 515.7373} C_DIS
LIN {X 55.9406,Y -120.1629,Z 156,A -66.528,B 21.269,C -0.7196,E1 21.3496,E2 514.1558} C_DIS
LIN {X 59.2658,Y -118.5597,Z 156,A -64.8278,B 21.2687,C -0.727,E1 21.3539,E2 512.4408} C_DIS
LIN {X 62.8389,Y -116.7055,Z 156,A -63.219,B 21.2688,C -0.7238,E1 21.3579,E2 510.8462} C_DIS
LIN {X 66.788,Y -114.4919,Z 156,A -61.1164,B 21.2685,C -0.734,E1 21.363,E2 508.7231} C_DIS
LIN {X 71.3174,Y -111.7261,Z 156,A -59.1493,B 21.2688,C -0.7231,E1 21.3676,E2 506.7936} C_DIS
LIN {X 73.9254,Y -110.0185,Z 156,A -57.6114,B 21.2685,C -0.7345,E1 21.3712,E2 505.2304} C_DIS
LIN {X 79.4146,Y -106.124,Z 156,A -54.9862,B 21.2687,C -0.7271,E1 21.3771,E2 502.6366} C_DIS
LIN {X 81.8295,Y -104.2727,Z 156,A -53.4662,B 21.2683,C -0.7395,E1 21.3805,E2 501.0894} C_DIS
LIN {X 85.2142,Y -101.5254,Z 156,A -51.3146,B 21.2678,C -0.7562,E1 21.3852,E2 498.9017} C_DIS
LIN {X 87.885,Y -99.2225,Z 156,A -49.9311,B 21.2678,C -0.753,E1 21.3881,E2 497.5336} C_DIS
LIN {X 91.642,Y -95.7634,Z 156,A -47.8851,B 21.2679,C -0.7505,E1 21.3922,E2 495.5045} C_DIS
LIN {X 94.8197,Y -92.6184,Z 156,A -45.7192,B 21.2674,C -0.7662,E1 21.3965,E2 493.3066} C_DIS
LIN {X 97.1048,Y -90.2195,Z 156,A -44.1475,B 21.2671,C -0.7763,E1 21.3995,E2 491.7154} C_DIS
LIN {X 99.8475,Y -87.1742,Z 156,A -42.9485,B 21.2678,C -0.7537,E1 21.4016,E2 490.5849} C_DIS
LIN {X 102.1489,Y -84.4659,Z 156,A -41.221,B 21.2674,C -0.7667,E1 21.4048,E2 488.8313} C_DIS
LIN {X 105.0205,Y -80.8686,Z 156,A -38.5361,B 21.266,C -0.8051,E1 21.4095,E2 486.0563} C_DIS
LIN {X 108.5228,Y -76.104,Z 156,A -36.8903,B 21.2673,C -0.7685,E1 21.412,E2 484.5202} C_DIS
LIN {X 110.391,Y -73.3674,Z 156,A -35.3062,B 21.2669,C -0.7797,E1 21.4145,E2 482.9149} C_DIS
LIN {X 112.6334,Y -69.8758,Z 156,A -33.5363,B 21.2669,C -0.7836,E1 21.4171,E2 481.145} C_DIS
LIN {X 114.8019,Y -66.2527,Z 156,A -31.7491,B 21.2667,C -0.787,E1 21.4197,E2 479.3595} C_DIS
LIN {X 116.7349,Y -62.7842,Z 156,A -29.9724,B 21.2664,C -0.7948,E1 21.4221,E2 477.5725} C_DIS
LIN {X 118.6902,Y -59.0012,Z 156,A -28.4241,B 21.2667,C -0.7863,E1 21.424,E2 476.0573} C_DIS
LIN {X 119.7249,Y -56.8718,Z 156,A -27.2406,B 21.2663,C -0.797,E1 21.4254,E2 474.8523} C_DIS
LIN {X 121.1559,Y -53.7564,Z 156,A -25.7032,B 21.2661,C -0.804,E1 21.4272,E2 473.3055} C_DIS
LIN {X 122.5185,Y -50.5756,Z 156,A -24.3466,B 21.2661,C -0.8019,E1 21.4287,E2 471.9636} C_DIS
LIN {X 123.9868,Y -46.8595,Z 156,A -22.7422,B 21.2661,C -0.8013,E1 21.4303,E2 470.3715} C_DIS
LIN {X 124.8313,Y -44.5611,Z 156,A -21.5133,B 21.2658,C -0.8127,E1 21.4315,E2 469.1197} C_DIS
LIN {X 126.1512,Y -40.6742,Z 156,A -19.3452,B 21.2649,C -0.837,E1 21.4334,E2 466.8997} C_DIS
LIN {X 127.2746,Y -37.0085,Z 156,A -18.0949,B 21.2654,C -0.8226,E1 21.4344,E2 465.6972} C_DIS
LIN {X 128.123,Y -33.955,Z 156,A -16.7667,B 21.2654,C -0.8249,E1 21.4353,E2 464.3719} C_DIS
LIN {X 128.9505,Y -30.6652,Z 156,A -15.0477,B 21.2647,C -0.8416,E1 21.4365,E2 462.6191} C_DIS
LIN {X 130.0492,Y -25.6163,Z 156,A -13.1214,B 21.265,C -0.834,E1 21.4375,E2 460.7272} C_DIS
LIN {X 130.7663,Y -21.6482,Z 156,A -11.4485,B 21.2649,C -0.8362,E1 21.4384,E2 459.0599} C_DIS
LIN {X 131.2128,Y -18.7528,Z 156,A -10.093,B 21.2646,C -0.8444,E1 21.4389,E2 457.6913} C_DIS
LIN {X 131.7024,Y -14.9481,Z 156,A -8.2056,B 21.264,C -0.8607,E1 21.4395,E2 455.7728} C_DIS
LIN {X 132.174,Y -9.9296,Z 156,A -6.267,B 21.2641,C -0.8562,E1 21.44,E2 453.8604} C_DIS
LIN {X 132.3849,Y -6.5384,Z 156,A -4.8082,B 21.264,C -0.8604,E1 21.4402,E2 452.4003} C_DIS
LIN {X 132.526,Y -2.3173,Z 156,A -3.0006,B 21.2638,C -0.8653,E1 21.4403,E2 450.5921} C_DIS
LIN {X 132.5386,Y 1.5641,Z 156,A -1.2321,B 21.2634,C -0.875,E1 21.4403,E2 448.8097} C_DIS
LIN {X 132.429,Y 5.5893,Z 156,A 0.4974,B 21.2632,C -0.88,E1 21.4401,E2 447.0787} C_DIS
LIN {X 132.1865,Y 9.7586,Z 156,A 2.1905,B 21.2632,C -0.8804,E1 21.4398,E2 445.3967} C_DIS
LIN {X 131.824,Y 13.8219,Z 156,A 3.9205,B 21.263,C -0.8844,E1 21.4394,E2 443.668} C_DIS
LIN {X 131.4961,Y 16.6602,Z 156,A 5.0339,B 21.2631,C -0.8824,E1 21.439,E2 442.5677} C_DIS
LIN {X 131.1665,Y 19.0762,Z 156,A 6.1313,B 21.2629,C -0.8878,E1 21.4386,E2 441.4633} C_DIS
LIN {X 130.6893,Y 22.1098,Z 156,A 7.5154,B 21.2626,C -0.8947,E1 21.4379,E2 440.0703} C_DIS
LIN {X 129.8192,Y 26.7492,Z 156,A 10.3934,B 21.2607,C -0.941,E1 21.4363,E2 437.0853} C_DIS
LIN {X 128.4248,Y 32.7952,Z 156,A 11.7937,B 21.2629,C -0.8881,E1 21.4355,E2 435.8396} C_DIS
LIN {X 127.742,Y 35.3624,Z 156,A 13.8417,B 21.261,C -0.9343,E1 21.4339,E2 433.6793} C_DIS
LIN {X 126.4833,Y 39.6348,Z 156,A 15.1997,B 21.2619,C -0.913,E1 21.4328,E2 432.3887} C_DIS
LIN {X 125.6631,Y 42.1576,Z 156,A 16.3647,B 21.2617,C -0.9173,E1 21.4318,E2 431.2198} C_DIS
LIN {X 124.6086,Y 45.179,Z 156,A 17.7649,B 21.2615,C -0.9222,E1 21.4305,E2 429.8157} C_DIS
LIN {X 123.4135,Y 48.3487,Z 156,A 19.2054,B 21.2614,C -0.9253,E1 21.429,E2 428.3762} C_DIS
LIN {X 122.1199,Y 51.5299,Z 156,A 20.6757,B 21.2612,C -0.9289,E1 21.4274,E2 426.9057} C_DIS
LIN {X 120.7495,Y 54.6652,Z 156,A 22.3075,B 21.2607,C -0.9403,E1 21.4256,E2 425.2533} C_DIS
LIN {X 119.1623,Y 58.0443,Z 156,A 23.6839,B 21.261,C -0.9336,E1 21.4239,E2 423.904} C_DIS
LIN {X 118.0095,Y 60.3504,Z 156,A 24.9111,B 21.2607,C -0.942,E1 21.4224,E2 422.6616} C_DIS
LIN {X 116.3584,Y 63.4791,Z 156,A 26.4349,B 21.2605,C -0.9459,E1 21.4203,E2 421.1368} C_DIS
LIN {X 114.2662,Y 67.1723,Z 156,A 28.2439,B 21.2604,C -0.9496,E1 21.4178,E2 419.3288} C_DIS
LIN {X 112.3283,Y 70.366,Z 156,A 29.8717,B 21.2601,C -0.9545,E1 21.4154,E2 417.6977} C_DIS
LIN {X 110.0118,Y 73.9354,Z 156,A 31.726,B 21.2599,C -0.9599,E1 21.4126,E2 415.8395} C_DIS
LIN {X 107.3595,Y 77.7355,Z 156,A 33.5405,B 21.2601,C -0.9561,E1 21.4097,E2 414.0461} C_DIS
LIN {X 105.1379,Y 80.7153,Z 156,A 35.3253,B 21.2595,C -0.9683,E1 21.4066,E2 412.2379} C_DIS
LIN {X 100.5112,Y 86.4083,Z 156,A 38.2205,B 21.2598,C -0.9629,E1 21.4016,E2 409.3735} C_DIS
LIN {X 97.6775,Y 89.5991,Z 156,A 40.2598,B 21.2592,C -0.9761,E1 21.3977,E2 407.3089} C_DIS
LIN {X 95.0023,Y 92.4313,Z 156,A 41.991,B 21.259,C -0.9819,E1 21.3943,E2 405.5706} C_DIS
LIN {X 91.8612,Y 95.5539,Z 156,A 44.5932,B 21.2573,C -1.018,E1 21.3889,E2 402.8824} C_DIS
LIN {X 87.5407,Y 99.5269,Z 156,A 46.3541,B 21.2587,C -0.9869,E1 21.3855,E2 401.2152} C_DIS
LIN {X 83.2479,Y 103.1438,Z 156,A 48.6522,B 21.2587,C -0.9857,E1 21.3806,E2 398.9311} C_DIS
LIN {X 80.4035,Y 105.3763,Z 156,A 50.3852,B 21.2583,C -0.9963,E1 21.3767,E2 397.1765} C_DIS
LIN {X 76.7457,Y 108.0701,Z 156,A 52.3663,B 21.2581,C -1.0005,E1 21.3722,E2 395.1923} C_DIS
LIN {X 73.0948,Y 110.5717,Z 156,A 54.2704,B 21.2581,C -1.0032,E1 21.3678,E2 393.2883} C_DIS
LIN {X 69.4117,Y 112.9199,Z 156,A 56.1221,B 21.2579,C -1.0045,E1 21.3634,E2 391.4402} C_DIS
LIN {X 65.7616,Y 115.0839,Z 156,A 57.9189,B 21.2579,C -1.0055,E1 21.3591,E2 389.6472} C_DIS
LIN {X 63.0616,Y 116.5858,Z 156,A 59.2889,B 21.2577,C -1.0089,E1 21.3557,E2 388.2726} C_DIS
LIN {X 59.7997,Y 118.2898,Z 156,A 60.8031,B 21.2578,C -1.0075,E1 21.352,E2 386.7672} C_DIS
LIN {X 56.7342,Y 119.7906,Z 156,A 62.2035,B 21.2578,C -1.0059,E1 21.3485,E2 385.3755} C_DIS
LIN {X 53.7969,Y 121.1378,Z 156,A 63.6349,B 21.2578,C -1.0091,E1 21.3448,E2 383.9397} C_DIS
LIN {X 50.3762,Y 122.6017,Z 156,A 65.371,B 21.2574,C -1.0166,E1 21.3403,E2 382.1878} C_DIS
LIN {X 46.5709,Y 124.0949,Z 156,A 66.7871,B 21.258,C -1.0026,E1 21.3367,E2 380.8139} C_DIS
LIN {X 44.5661,Y 124.8295,Z 156,A 67.8825,B 21.2576,C -1.0112,E1 21.3338,E2 379.6976} C_DIS
LIN {X 41.1816,Y 125.9881,Z 156,A 69.452,B 21.2576,C -1.0135,E1 21.3296,E2 378.1253} C_DIS
LIN {X 37.9514,Y 126.9986,Z 156,A 71.2873,B 21.2567,C -1.0313,E1 21.3246,E2 376.2449} C_DIS
LIN {X 34.6178,Y 127.9463,Z 156,A 72.2848,B 21.2577,C -1.01,E1 21.3221,E2 375.308} C_DIS
LIN {X 30.1419,Y 129.0748,Z 156,A 74.4473,B 21.2573,C -1.0186,E1 21.3162,E2 373.1257} C_DIS
LIN {X 26.8473,Y 129.7992,Z 156,A 75.7642,B 21.2576,C -1.0131,E1 21.3126,E2 371.8259} C_DIS
LIN {X 23.4981,Y 130.4466,Z 156,A 77.384,B 21.2572,C -1.0202,E1 21.3081,E2 370.1889} C_DIS
LIN {X 19.5234,Y 131.1025,Z 156,A 79.2748,B 21.2569,C -1.0273,E1 21.3028,E2 368.2806} C_DIS
LIN {X 15.0964,Y 131.685,Z 156,A 80.9884,B 21.2573,C -1.0182,E1 21.2982,E2 366.5937} C_DIS
LIN {X 12.2061,Y 131.9837,Z 156,A 82.2007,B 21.2574,C -1.0165,E1 21.2948,E2 365.3871} C_DIS
LIN {X 8.9514,Y 132.2454,Z 156,A 83.7957,B 21.257,C -1.0247,E1 21.2903,E2 363.7704} C_DIS
LIN {X 5.1523,Y 132.446,Z 156,A 85.4441,B 21.257,C -1.0248,E1 21.2857,E2 362.1223} C_DIS
LIN {X 1.008,Y 132.5427,Z 156,A 87.158,B 21.2572,C -1.0212,E1 21.281,E2 360.4186} C_DIS
LIN {X -2.5848,Y 132.5216,Z 156,A 88.7955,B 21.257,C -1.0246,E1 21.2764,E2 358.7717} C_DIS
LIN {X -6.6701,Y 132.3783,Z 156,A 90.4145,B 21.2574,C -1.0176,E1 21.2719,E2 357.1716} C_DIS
LIN {X -10.0915,Y 132.1622,Z 156,A 92.1721,B 21.2568,C -1.029,E1 21.2669,E2 355.3816} C_DIS
LIN {X -14.0925,Y 131.7948,Z 156,A 93.7424,B 21.2572,C -1.021,E1 21.2626,E2 353.8326} C_DIS
LIN {X -18.1878,Y 131.2935,Z 156,A 95.5396,B 21.2572,C -1.0205,E1 21.2576,E2 352.0351} C_DIS
LIN {X -21.97,Y 130.7126,Z 156,A 97.2665,B 21.2572,C -1.0226,E1 21.2528,E2 350.3005} C_DIS
LIN {X -25.4456,Y 130.0818,Z 156,A 98.6624,B 21.2574,C -1.0158,E1 21.2491,E2 348.9216} C_DIS
LIN {X -33.78,Y 128.1697,Z 156,A 102.1638,B 21.258,C -1.0041,E1 21.2396,E2 345.4469} C_DIS
LIN {X -39.276,Y 126.5941,Z 156,A 104.768,B 21.2578,C -1.0071,E1 21.2326,E2 342.8292} C_DIS
LIN {X -42.6502,Y 125.499,Z 156,A 106.345,B 21.2578,C -1.0071,E1 21.2284,E2 341.2486} C_DIS
LIN {X -45.1754,Y 124.6099,Z 156,A 107.5452,B 21.2578,C -1.0076,E1 21.2252,E2 340.0443} C_DIS
LIN {X -48.9415,Y 123.1809,Z 156,A 109.9292,B 21.2567,C -1.0327,E1 21.2189,E2 337.5849} C_DIS
LIN {X -53.6334,Y 121.211,Z 156,A 111.3514,B 21.2583,C -0.9965,E1 21.2155,E2 336.2586} C_DIS
LIN {X -57.3502,Y 119.4963,Z 156,A 113.6335,B 21.2574,C -1.0155,E1 21.2096,E2 333.917} C_DIS
LIN {X -60.7369,Y 117.8127,Z 156,A 115.0304,B 21.258,C -1.0028,E1 21.2062,E2 332.5507} C_DIS
LIN {X -64.295,Y 115.9096,Z 156,A 116.6872,B 21.2583,C -0.9963,E1 21.2021,E2 330.9066} C_DIS
LIN {X -68.0276,Y 113.7592,Z 156,A 118.5763,B 21.2584,C -0.9941,E1 21.1976,E2 329.0165} C_DIS
LIN {X -71.7393,Y 111.456,Z 156,A 120.5138,B 21.2584,C -0.9927,E1 21.193,E2 327.0756} C_DIS
LIN {X -75.4379,Y 108.9867,Z 156,A 122.4731,B 21.2586,C -0.9906,E1 21.1885,E2 325.1143} C_DIS
LIN {X -79.1762,Y 106.3015,Z 156,A 124.4086,B 21.2588,C -0.9843,E1 21.1841,E2 323.1879} C_DIS
LIN {X -82.4537,Y 103.7799,Z 156,A 126.2292,B 21.2589,C -0.982,E1 21.1801,E2 321.3659} C_DIS
LIN {X -85.9029,Y 100.9434,Z 156,A 128.1663,B 21.2591,C -0.9781,E1 21.176,E2 319.4307} C_DIS
LIN {X -89.2939,Y 97.957,Z 156,A 130.1235,B 21.2593,C -0.9738,E1 21.1719,E2 317.4758} C_DIS
LIN {X -92.2811,Y 95.1477,Z 156,A 131.9273,B 21.2594,C -0.971,E1 21.1683,E2 315.6709} C_DIS
LIN {X -95.4707,Y 91.9475,Z 156,A 133.8745,B 21.2596,C -0.9661,E1 21.1645,E2 313.7274} C_DIS
LIN {X -98.3172,Y 88.8968,Z 156,A 135.6789,B 21.2598,C -0.9617,E1 21.1611,E2 311.9256} C_DIS
LIN {X -101.2317,Y 85.5637,Z 156,A 137.6638,B 21.2599,C -0.9598,E1 21.1574,E2 309.9352} C_DIS
LIN {X -104.0739,Y 82.0827,Z 156,A 139.603,B 21.2601,C -0.9546,E1 21.1541,E2 307.9994} C_DIS
LIN {X -106.7404,Y 78.5835,Z 156,A 141.4686,B 21.2604,C -0.9481,E1 21.1509,E2 306.1411} C_DIS
LIN {X -109.0932,Y 75.2838,Z 156,A 143.2777,B 21.2605,C -0.9457,E1 21.148,E2 304.328} C_DIS
LIN {X -111.5264,Y 71.6294,Z 156,A 145.1509,B 21.2608,C -0.9395,E1 21.1452,E2 302.4608} C_DIS
LIN {X -113.602,Y 68.2905,Z 156,A 146.8357,B 21.261,C -0.9341,E1 21.1427,E2 300.7806} C_DIS
LIN {X -115.6329,Y 64.7916,Z 156,A 148.7269,B 21.261,C -0.935,E1 21.1401,E2 298.8751} C_DIS
LIN {X -117.8457,Y 60.6721,Z 156,A 150.4885,B 21.2617,C -0.9186,E1 21.1379,E2 297.1479} C_DIS
LIN {X -118.9982,Y 58.377,Z 156,A 151.6494,B 21.2617,C -0.9174,E1 21.1364,E2 295.9829} C_DIS
LIN {X -120.6726,Y 54.837,Z 156,A 153.3828,B 21.2618,C -0.914,E1 21.1344,E2 294.2474} C_DIS
LIN {X -121.774,Y 52.3407,Z 156,A 154.5903,B 21.2619,C -0.9117,E1 21.133,E2 293.0385} C_DIS
LIN {X -122.9021,Y 49.6331,Z 156,A 155.8843,B 21.262,C -0.9089,E1 21.1317,E2 291.7435} C_DIS
LIN {X -124.1678,Y 46.3761,Z 156,A 157.3692,B 21.2623,C -0.9033,E1 21.1302,E2 290.2642} C_DIS
LIN {X -125.2737,Y 43.3,Z 156,A 158.8001,B 21.2624,C -0.8997,E1 21.1289,E2 288.8336} C_DIS
LIN {X -126.2786,Y 40.2754,Z 156,A 160.2733,B 21.2624,C -0.8993,E1 21.1276,E2 287.3513} C_DIS
LIN {X -127.3552,Y 36.7332,Z 156,A 161.7332,B 21.2629,C -0.8886,E1 21.1264,E2 285.9109} C_DIS
LIN {X -128.1006,Y 34.0392,Z 156,A 163.0504,B 21.2629,C -0.8893,E1 21.1255,E2 284.5827} C_DIS
LIN {X -129.0414,Y 30.2879,Z 156,A 164.6981,B 21.2631,C -0.8831,E1 21.1244,E2 282.9408} C_DIS
LIN {X -129.5854,Y 27.8578,Z 156,A 165.885,B 21.2631,C -0.8842,E1 21.1237,E2 281.7424} C_DIS
LIN {X -131.0946,Y 19.5746,Z 156,A 169.5926,B 21.2634,C -0.8753,E1 21.1219,E2 278.0329} C_DIS
LIN {X -131.7632,Y 14.3868,Z 156,A 171.696,B 21.2639,C -0.8618,E1 21.1212,E2 275.9521} C_DIS
LIN {X -132.0229,Y 11.7827,Z 156,A 172.8087,B 21.2641,C -0.8574,E1 21.1209,E2 274.8435} C_DIS
LIN {X -132.2577,Y 8.7611,Z 156,A 174.2493,B 21.2641,C -0.8585,E1 21.1206,E2 273.3895} C_DIS
LIN {X -132.4471,Y 5.1239,Z 156,A 175.8135,B 21.2643,C -0.8531,E1 21.1204,E2 271.829} C_DIS
LIN {X -132.5452,Y 0.5395,Z 156,A 177.6433,B 21.2647,C -0.8406,E1 21.1204,E2 270.0208} C_DIS
LIN {X -132.5291,Y -2.1326,Z 156,A 179.2965,B 21.2641,C -0.8572,E1 21.1204,E2 268.3095} C_DIS
LIN {X -132.429,Y -5.5883,Z 156,A -179.5783,B 21.2648,C -0.8374,E1 21.1205,E2 267.2312} C_DIS
LIN {X -132.2396,Y -9.0311,Z 156,A -177.5678,B 21.2642,C -0.8539,E1 21.1209,E2 265.1604} C_DIS
LIN {X -131.9062,Y -13.0139,Z 156,A -176.2748,B 21.2651,C -0.8307,E1 21.1213,E2 263.9225} C_DIS
LIN {X -131.1545,Y -19.1606,Z 156,A -173.6221,B 21.2654,C -0.8213,E1 21.1222,E2 261.2769} C_DIS
LIN {X -130.7901,Y -21.5057,Z 156,A -171.9106,B 21.2645,C -0.8462,E1 21.123,E2 259.4841} C_DIS
LIN {X -129.887,Y -26.416,Z 156,A -170.6518,B 21.2661,C -0.8027,E1 21.1237,E2 258.3372} C_DIS
LIN {X -129.4431,Y -28.5169,Z 156,A -169.4879,B 21.2659,C -0.8094,E1 21.1243,E2 257.1464} C_DIS
LIN {X -128.799,Y -31.2939,Z 156,A -168.2319,B 21.2659,C -0.8066,E1 21.1252,E2 255.8893} C_DIS
LIN {X -127.9774,Y -34.501,Z 156,A -166.71,B 21.266,C -0.806,E1 21.1262,E2 254.3585} C_DIS
LIN {X -127.0113,Y -37.9079,Z 156,A -165.2588,B 21.2663,C -0.7981,E1 21.1274,E2 252.919} C_DIS
LIN {X -126.2322,Y -40.4207,Z 156,A -164.0661,B 21.2663,C -0.797,E1 21.1284,E2 251.7213} C_DIS
LIN {X -125.1603,Y -43.6272,Z 156,A -162.1235,B 21.2658,C -0.8125,E1 21.1302,E2 249.7223} C_DIS
LIN {X -123.7159,Y -47.5709,Z 156,A -160.913,B 21.2668,C -0.7823,E1 21.1313,E2 248.5875} C_DIS
LIN {X -122.7758,Y -49.9466,Z 156,A -159.6763,B 21.2668,C -0.7845,E1 21.1326,E2 247.3364} C_DIS
LIN {X -121.3032,Y -53.4272,Z 156,A -157.5948,B 21.2663,C -0.7984,E1 21.135,E2 245.2028} C_DIS
LIN {X -119.7467,Y -56.826,Z 156,A -156.583,B 21.2673,C -0.7689,E1 21.1361,E2 244.2661} C_DIS
LIN {X -118.7052,Y -58.9709,Z 156,A -155.3651,B 21.2671,C -0.7738,E1 21.1376,E2 243.0269} C_DIS
LIN {X -117.1985,Y -61.9109,Z 156,A -153.9024,B 21.2672,C -0.7713,E1 21.1395,E2 241.5617} C_DIS
LIN {X -114.9344,Y -66.0236,Z 156,A -151.8837,B 21.2674,C -0.7654,E1 21.1423,E2 239.5468} C_DIS
LIN {X -113.1518,Y -69.0337,Z 156,A -150.2403,B 21.2674,C -0.7668,E1 21.1447,E2 237.8891} C_DIS
LIN {X -110.4279,Y -73.3121,Z 156,A -148.2267,B 21.2678,C -0.7538,E1 21.1477,E2 235.8996} C_DIS
LIN {X -108.5228,Y -76.104,Z 156,A -146.5345,B 21.2676,C -0.7597,E1 21.1504,E2 234.181} C_DIS
LIN {X -105.8019,Y -79.8425,Z 156,A -144.7561,B 21.2681,C -0.7456,E1 21.1533,E2 232.4313} C_DIS
LIN {X -103.7928,Y -82.4376,Z 156,A -143.1925,B 21.2681,C -0.7483,E1 21.156,E2 230.8514} C_DIS
LIN {X -101.2819,Y -85.5045,Z 156,A -141.3915,B 21.2681,C -0.748,E1 21.1593,E2 229.0414} C_DIS
LIN {X -98.3713,Y -88.8372,Z 156,A -139.497,B 21.2681,C -0.7429,E1 21.1628,E2 227.1508} C_DIS
LIN {X -95.4993,Y -91.918,Z 156,A -137.5892,B 21.2682,C -0.7426,E1 21.1665,E2 225.2339} C_DIS
LIN {X -92.3725,Y -95.0592,Z 156,A -135.9219,B 21.2687,C -0.7281,E1 21.1697,E2 223.5983} C_DIS
LIN {X -89.9333,Y -97.3703,Z 156,A -134.2433,B 21.2685,C -0.7347,E1 21.1732,E2 221.8933} C_DIS
LIN {X -86.5388,Y -100.3987,Z 156,A -132.3293,B 21.2687,C -0.7286,E1 21.1772,E2 219.9871} C_DIS
LIN {X -83.3987,Y -103.0222,Z 156,A -130.5349,B 21.2687,C -0.7264,E1 21.1811,E2 218.1906} C_DIS
LIN {X -80.0836,Y -105.62,Z 156,A -128.6695,B 21.2687,C -0.7251,E1 21.1852,E2 216.3209} C_DIS
LIN {X -76.4598,Y -108.2718,Z 156,A -126.7692,B 21.2689,C -0.72,E1 21.1895,E2 214.4266} C_DIS
LIN {X -72.9973,Y -110.6358,Z 156,A -124.9068,B 21.2689,C -0.7193,E1 21.1938,E2 212.5589} C_DIS
LIN {X -69.0143,Y -113.1637,Z 156,A -122.811,B 21.2689,C -0.7186,E1 21.1988,E2 210.457} C_DIS
LIN {X -65.0276,Y -115.5002,Z 156,A -120.8663,B 21.2692,C -0.7135,E1 21.2035,E2 208.5195} C_DIS
LIN {X -60.8795,Y -117.7401,Z 156,A -118.9286,B 21.2694,C -0.7065,E1 21.2083,E2 206.5948} C_DIS
LIN {X -58.4468,Y -118.9637,Z 156,A -117.7202,B 21.2694,C -0.7065,E1 21.2113,E2 205.3828} C_DIS
LIN {X -55.2838,Y -120.4666,Z 156,A -116.2506,B 21.2694,C -0.7027,E1 21.215,E2 203.919} C_DIS
LIN {X -52.0106,Y -121.9167,Z 156,A -114.4565,B 21.2692,C -0.7117,E1 21.2197,E2 202.0949} C_DIS
LIN {X -47.9493,Y -123.5688,Z 156,A -112.7668,B 21.2696,C -0.701,E1 21.224,E2 200.4307} C_DIS
LIN {X -44.2639,Y -124.9385,Z 156,A -111.0833,B 21.2696,C -0.6987,E1 21.2284,E2 198.7493} C_DIS
LIN {X -41.1249,Y -126.007,Z 156,A -109.3449,B 21.2692,C -0.7109,E1 21.2331,E2 196.9735} C_DIS
LIN {X -36.5423,Y -127.4111,Z 156,A -107.2581,B 21.2692,C -0.7101,E1 21.2387,E2 194.8848} C_DIS
LIN {X -33.4357,Y -128.2611,Z 156,A -106.1728,B 21.2697,C -0.6957,E1 21.2416,E2 193.8373} C_DIS
LIN {X -30.0882,Y -129.0871,Z 156,A -104.6127,B 21.2697,C -0.698,E1 21.2458,E2 192.2684} C_DIS
LIN {X -26.5096,Y -129.8679,Z 156,A -103.0596,B 21.2697,C -0.6959,E1 21.25,E2 190.7187} C_DIS
LIN {X -22.8235,Y -130.5673,Z 156,A -101.3251,B 21.2696,C -0.7003,E1 21.2549,E2 188.97} C_DIS
LIN {X -18.1111,Y -131.3045,Z 156,A -99.448,B 21.2698,C -0.6915,E1 21.26,E2 187.1152} C_DIS
LIN {X -14.8366,Y -131.7148,Z 156,A -97.867,B 21.2696,C -0.6982,E1 21.2644,E2 185.5147} C_DIS
LIN {X -11.0646,Y -132.0835,Z 156,A -96.3243,B 21.2698,C -0.6938,E1 21.2687,E2 183.9831} C_DIS
LIN {X -7.0566,Y -132.3588,Z 156,A -94.5561,B 21.2698,C -0.6952,E1 21.2736,E2 182.2103} C_DIS
LIN {X -3.455,Y -132.5014,Z 156,A -92.956,B 21.2697,C -0.6972,E1 21.2781,E2 180.6044} C_DIS
LIN {X 0.9151,Y -132.5419,Z 156,A -91.2205,B 21.2699,C -0.6907,E1 21.2829,E2 178.8869} C_DIS
Enddeposition()
LIN {X 0.9151,Y -132.5419,Z 156,A -91.2205,B 21.2699,C -0.6907,E1 21.2829,E2 178.8869} C_DIS
Startdeposition()
$VEL.CP = VEL_PRINT
LIN {X 0.4793,Y -131.6119,Z 156,A -91.78,B 20.2007,C -0.5199,E1 20.2068,E2 179.8207} C_DIS
LIN {X -3.7388,Y -131.5594,Z 156,A -93.5214,B 20.2006,C -0.5236,E1 20.202,E2 181.5516} C_DIS
LIN {X -7.8159,Y -131.3804,Z 156,A -95.321,B 20.2006,C -0.5225,E1 20.1969,E2 183.3547} C_DIS
LIN {X -11.5185,Y -131.1081,Z 156,A -97.0221,B 20.2007,C -0.5191,E1 20.1922,E2 185.0666} C_DIS
LIN {X -15.349,Y -130.7145,Z 156,A -98.3839,B 20.2004,C -0.5324,E1 20.1885,E2 186.3911} C_DIS
LIN {X -21.2999,Y -129.8778,Z 156,A -101.2437,B 20.2006,C -0.523,E1 20.1805,E2 189.281} C_DIS
LIN {X -24.7343,Y -129.2671,Z 156,A -102.7239,B 20.2006,C -0.5251,E1 20.1764,E2 190.7569} C_DIS
LIN {X -28.0649,Y -128.5855,Z 156,A -104.2171,B 20.2006,C -0.5253,E1 20.1724,E2 192.2519} C_DIS
LIN {X -31.665,Y -127.7471,Z 156,A -106.125,B 20.2008,C -0.514,E1 20.1671,E2 194.1957} C_DIS
LIN {X -34.8739,Y -126.9091,Z 156,A -107.2916,B 20.2005,C -0.5262,E1 20.164,E2 195.3293} C_DIS
LIN {X -37.9997,Y -126.0081,Z 156,A -108.9142,B 20.2007,C -0.5189,E1 20.1596,E2 196.9767} C_DIS
LIN {X -42.8395,Y -124.4451,Z 156,A -110.9629,B 20.2005,C -0.5273,E1 20.1542,E2 199.0056} C_DIS
LIN {X -46.4708,Y -123.1353,Z 156,A -112.6029,B 20.2005,C -0.5305,E1 20.15,E2 200.6407} C_DIS
LIN {X -52.1679,Y -120.8314,Z 156,A -115.2633,B 20.2003,C -0.5338,E1 20.1431,E2 203.2989} C_DIS
LIN {X -55.1191,Y -119.514,Z 156,A -116.6757,B 20.2003,C -0.5352,E1 20.1395,E2 204.7117} C_DIS
LIN {X -57.9301,Y -118.1774,Z 156,A -118.0717,B 20.2003,C -0.5352,E1 20.136,E2 206.1123} C_DIS
LIN {X -60.7581,Y -116.7492,Z 156,A -119.4599,B 20.2003,C -0.5366,E1 20.1325,E2 207.5012} C_DIS
Enddeposition()
END
